(* Logix 5000 project; controller RSL5k_18_Template_noLib Emulate 5570 rev 32.11; software revision 32.02; part 12 of 16 *)
(* tags used below, declared in another part *)
   Inp_SpeedFdbk : REAL;   // Speed Feedbak in Drive Units (typ. 0-32767 = 0 to max freq.)
   Inp_Datalink : REAL;   // Auxiliary Signal (datalink) Input in Drive (raw) Units
   Inp_Ready : BOOL;   // 1=Drive is ready to run
   Inp_Running : BOOL;   // 1=Drive is Running (active)
   Inp_CommandDir : BOOL;   // 1=Drive is commanded Forward, 0=Drive is commanded Reverse
   Inp_ActualDir : BOOL;   // 1=Drive is running Forward, 0=Drive is running Reverse
   Inp_Accelerating : BOOL;   // 1=Drive is accelerating
   Inp_Decelerating : BOOL;   // 1=Drive is decelerating
   Inp_Alarm : BOOL;   // 1=Drive has an Alarm Condition (see drive display or manual)
   Inp_AtSpeed : BOOL;   // 1=Drive is at commanded speed
   Inp_IOFault : BOOL;   // Input Communication Status 0=OK, 1=fail
   Inp_Sim : BOOL;   // 1=Simulate working drive; 0=Start/Stop/ Monitor actual drive
   Inp_OvrdSpeed : REAL;   // Value to set Speed Reference in Override Mode (SpeedRef EU)
   Inp_OvrdOutDatalink : REAL;   // Value to set Output Datalink in Override Mode (OutDatalink EU)
   Inp_HornInh : BOOL;   // 1 = Inhibit audible alert, 0 = Alllow audible alert
   Inp_Reset : BOOL;   // 1=Reset Shed Latches and Cleared Alarms
   Cfg_HasJog : BOOL;   // 1=Drive Jog Command enabled/visible, 0=Drive Jog Command not allowed
   Cfg_AllowLocal : BOOL;   // 1=Allow Local Start/Stop without alarm, 0=Start/Stop from HMI/prog only
   Cfg_HasRunFdbk : BOOL;   // 1=Drive provides feedback signal on Inp_Running when running
   Cfg_UseRunFdbk : BOOL;   // 1=Drive run feedback should be used for failure checking
   Cfg_HasSpeedFdbk : BOOL;   // 1=Drive provides speed feedback on Inp_SpeedFdbk
   Cfg_UseSpeedFdbk : BOOL;   // 1=Drive speed determines running state, 0=state determined by drive Active input bit
   Cfg_HasInpDatalink : BOOL;   // 1=A signal is connected to Inp_Datalink
   Cfg_HasOutDatalink : BOOL;   // 1=A signal is connected to Out_Datalink
   Cfg_HasMoreObj : BOOL;   // 1=Tells HMI an object with more info is available
   Cfg_SetTrack : BOOL;   // 1=Settings track for unselected sources, 0=no tracking
   Cfg_SetTrackOvrdHand : BOOL;   // 1=Prog/Oper/Ext Settings track Override/Hand
   Cfg_OCmdResets : BOOL;   // 1=New drive OCmd resets shed latches and cleared alarms, 0=OCmdReset req'd.
   Cfg_XCmdResets : BOOL;   // 1=New drive XCmd resets shed latches and cleared alarms, 0=XCmdReset req'd.
   Cfg_OvrdPermIntlk : BOOL;   // 1=Override ignores Bypassable Perm/ Intlk; 0=always use Perm/Intlk
   Cfg_SimScaleEU : BOOL;   // 1=In simulation, scale Speed Ref EU to Speed Fdbk EU
   Cfg_SimScaleRaw : BOOL;   // 1=In simulation, scale Speed Ref EU to raw, then raw to Speed Fdbk EU
   Cfg_DecPlcs : DINT;   // Number of decimal places for speed ref/fdbk display (0..6)
   Cfg_InpDLDecPlcs : DINT;   // Number of decimal places for Input Datalink display (0..6)
   Cfg_OutDLDecPlcs : DINT;   // Number of decimal places for Output Datalink display (0..6)
   Cfg_MinSpdRef : REAL;   // Minimum Speed Reference in EU (for limiting)
   Cfg_MaxSpdRef : REAL;   // Maximum Speed Reference in EU (for limiting)
   Cfg_SpeedRefRawMin : REAL;   // Speed Reference Minimum in Drive (raw) Units (for scaling)
   Cfg_SpeedRefRawMax : REAL;   // Speed Reference Maximum in Drive (raw) Units (for scaling)
   Cfg_SpeedRefEUMin : REAL;   // Speed Reference Minimum in Engineering Units (for scaling)
   Cfg_SpeedRefEUMax : REAL;   // Speed Reference Maximum in Engineering Units (for scaling)
   Cfg_SpeedFdbkRawMin : REAL;   // Speed Feedback Minimum in Drive (raw) Units (for scaling)
   Cfg_SpeedFdbkRawMax : REAL;   // Speed Feedback Maximum in Drive (raw) Units (for scaling)
   Cfg_SpeedFdbkEUMin : REAL;   // Speed Feedback Minimum in Engineering Units (for scaling)
   Cfg_SpeedFdbkEUMax : REAL;   // Speed Feedback Maximum in Engineering Units (for scaling)
   Cfg_InpDatalinkRawMin : REAL;   // Input Datalink Minimum in Drive (raw) Units (for scaling)
   Cfg_InpDatalinkRawMax : REAL;   // Input Datalink Maximum in Drive (raw) Units (for scaling)
   Cfg_InpDatalinkEUMin : REAL;   // Input Datalink Minimum in Engineering Units (for scaling)
   Cfg_InpDatalinkEUMax : REAL;   // Input Datalink Maximum in Engineering Units (for scaling)
   Cfg_OutDatalinkMin : REAL;   // Minimum Output Datalink in EU (for limiting)
   Cfg_OutDatalinkMax : REAL;   // Maximum Output Datalink in EU (for limiting)
   Cfg_OutDatalinkRawMin : REAL;   // Output Datalink Minimum in Drive (raw) Units (for scaling)
   Cfg_OutDatalinkRawMax : REAL;   // Output Datalink Maximum in Drive (raw) Units (for scaling)
   Cfg_OutDatalinkEUMin : REAL;   // Output Datalink Minimum in Engineering Units (for scaling)
   Cfg_OutDatalinkEUMax : REAL;   // Output Datalink Maximum in Engineering Units (for scaling)
   Cfg_StartHornT : REAL;   // Time to sound audible on commanded start (sec) (0=disabled)
   Cfg_SimRampT : REAL;   // Time to ramp speed fdbk when in Simulation (sec)
   Cfg_FailToStartT : REAL;   // Time after Start to get Run Feedback before Fault (sec)
   Cfg_FailToStopT : REAL;   // Time after Stop to drop Run Feedback before Fault (sec)
   Cfg_ResetPulseT : REAL;   // Time to pulse Out_Reset to clear drive fault
   Cfg_MaxJogT : REAL;   // Maximum jog time (sec, 0=unlimited)
   Cfg_OperKeep : SINT;   // Oper keeps control in Prog / Ext: .0=Reference, .1=Start/Stop/Fwd/ Rev, .3=OutDatalink
   Cfg_ProgKeep : SINT;   // Prog keeps control in Oper / Ext: .0=Reference, .1=Start/Stop/Fwd/ Rev, .3=OutDatalink
   Cfg_ExtKeep : SINT;   // Ext keeps control in Prog / Oper: .0=Reference, .1=Start/Stop/Fwd/ Rev, .3=OutDatalink
   PSet_SpeedRef : REAL;   // Program Setting of Speed Reference (EU)
   PSet_OutDatalink : REAL;   // Program Setting of Output Datalink (EU)
   PSet_Owner : DINT;   // Program Owner Request ID (non-zero) or Release (zero)
   XSet_SpeedRef : REAL;   // External Setting of Speed Reference (EU)
   XSet_OutDatalink : REAL;   // External Setting of Output Datalink (EU)
   PCmd_Reset : BOOL;   // Program Command to Reset drive fault and all Alarms requiring Reset
   PCmd_FailToStartAck : ALIAS FOR FailToStart.PCmd_Ack;   // Program Command to Acknowledge Fail to Start Alarm
   PCmd_FailToStopAck : ALIAS FOR FailToStop.PCmd_Ack;   // Program Command to Acknowledge Fail to Stop Alarm
   PCmd_IntlkTripAck : ALIAS FOR IntlkTrip.PCmd_Ack;   // Program Command to Acknowledge Interlock Trip Alarm
   PCmd_DriveFaultAck : ALIAS FOR DriveFault.PCmd_Ack;   // Program Command to Acknowledge Drive Fault Alarm
   PCmd_IOFaultAck : ALIAS FOR IOFault.PCmd_Ack;   // Program Command to Acknowledge I/O Fault Alarm
   XCmd_StartFwd : BOOL;   // External Command to Start Drive Forward
   XCmd_StartRev : BOOL;   // External Command to Start Drive Reverse
   XCmd_Stop : BOOL;   // External Command to Stop Drive
   XCmd_JogFwd : BOOL;   // External Command to Jog Drive Forward
   XCmd_JogRev : BOOL;   // External Command to Jog Drive Reverse
   XCmd_Reset : BOOL;   // Ext Cmd to clear shed latches and cleared alarms
   Val_SpeedFdbk : REAL;   // Speed Feedback (actual) from drive
   Val_InpDatalink : REAL;   // Input Datalink value from drive
   Val_SpeedRefEUMin : REAL;   // Minimum of Speed Reference = MIN (Cfg_SpeedFdbkEUMin, Cfg_SpeedFdbkEUMax)
   Val_SpeedRefEUMax : REAL;   // Maximum of Speed Reference = MAX (Cfg_SpeedFdbkEUMin, Cfg_SpeedFdbkEUMax)
   Val_SpeedFdbkEUMin : REAL;   // Minimum of Speed Feedback = MIN (Cfg_SpeedFdbkEUMin, Cfg_SpeedFdbkEUMax)
   Val_SpeedFdbkEUMax : REAL;   // Maximum of Speed Feedback = MAX (Cfg_SpeedFdbkEUMin, Cfg_SpeedFdbkEUMax)
   Val_Fdbk : DINT;   // Device Feedback 0=Stopped, 1=Running Fwd 2=Running Rev 3=Accelerating 4=Decelerating
   Val_Sts : DINT;   // Device Sts: 0=? 1=Stopped 2=RunFwd 3=RunRev 4=RunSlow 5=StartFwd 6=StartRev 7=StartSlow 8=JogFwd 9=JogRev 10=Stopping
   Val_Owner : DINT;   // Current Object Owner ID (0=not owned)
   Sts_CommandDir : BOOL;   // 1=Drive commanded to Forward, 0=Reverse
   Sts_ActualDir : BOOL;   // 1=Drive Actual direction is Forward, 0=Reverse
   Sts_Accel : BOOL;   // 1=Drive is Accelerating
   Sts_Decel : BOOL;   // 1=Drive is Decelerating
   Sts_NotReady : BOOL;   // 1=Drive is Not Ready (cannot be started) Check alarms, stops, faults
   Sts_Alarm : BOOL;   // 1=Drive has an Alarm (see drive display or manual)
   Sts_AtSpeed : BOOL;   // 1=Drive is running at reference speed
   Sts_Bypass : BOOL;   // 1=Bypassable Interlocks and Permissives are Bypassed
   Sts_BypActive : BOOL;   // 1=Bypassing Active (Bypassed or Maintenance)
   Nrdy_CfgErr : BOOL;   // 1=Device Not Ready: Configuration Error
   Nrdy_Fail : BOOL;   // 1=Device Not Ready: Device Failure (Shed Requires Reset)
   Nrdy_IOFault : BOOL;   // 1=Device Not Ready: I/O Fault (Shed Requires Reset)
   Nrdy_PrioStop : BOOL;   // 1=Device Not Ready: Oper/Ext Priority Stop Requires Reset
   Sts_MaintByp : BOOL;   // 1=A Maintenance Bypass is Active, display icon
   Err_Timer : BOOL;   // 1=Error in Config: Invalid Check or Reset Pulse Time (use 0 to 2147483)
   Err_Sim : BOOL;   // 1=Error in Config: simulation timer preset: use 0 to 2147483)
   Err_FdbkRaw : BOOL;   // 1=Erron in Config: Speed Fdbk Raw Min = Max
   Err_FdbkEU : BOOL;   // 1=Error in Config: Speed Fdbk EU Min = Max
   Err_RefLim : BOOL;   // 1=Error in Config: Speed Ref Limit Min > Max
   Err_RefEU : BOOL;   // 1=Error in Config: Speed Ref EU Min = Max
   Err_RefRaw : BOOL;   // 1=Error in Config: Speed Ref Raw Min = Max
   Err_InpDLRaw : BOOL;   // 1=Error in Config: Input Datalink Raw Min = Max
   Err_InpDLEU : BOOL;   // 1=Error in Config: Input Datalink EU Min = Max
   Err_OutDLLim : BOOL;   // 1=Error in Config: Output Datalink Limits Min > Max
   Err_OutDLEU : BOOL;   // 1=Error in Config: Output Datalink EU Min = Max
   Err_OutDLRaw : BOOL;   // 1=Error in Config: Output Datalink Raw Min = Max
   Sts_Hand : ALIAS FOR CmdSrc.Sts_Hand;
   Sts_Maint : ALIAS FOR CmdSrc.Sts_Maint;
   Sts_Ovrd : ALIAS FOR CmdSrc.Sts_Ovrd;
   Sts_Ext : ALIAS FOR CmdSrc.Sts_Ext;
   Sts_Prog : ALIAS FOR CmdSrc.Sts_Prog;
   Sts_Oper : ALIAS FOR CmdSrc.Sts_Oper;
   Sts_RdyAck : BOOL;   // 1=An alarm is ready to be acknowledged
   Sts_FailToStart : ALIAS FOR FailToStart.Inp;   // 1=Drive Failed to Start (One-Shot)
   Sts_FailToStop : ALIAS FOR FailToStop.Inp;   // 1=Drive Failed to Stop
   P_VSD : BOOL;   // Unique Parameter Name for auto - discovery
   CmdSrc : P_CmdSrc;   // Drive Mode Selection
   IOFault : P_Alarm;   // I/O Fault Alarm
   IntlkTrip : P_Alarm;   // Interlock Trip Alarm
   FailToStop : P_Alarm;   // Drive Failed to Stop Alarm
   FailToStart : P_Alarm;   // Drive Failed to Start Alarm
   Cfg_Tag : STRING_20;   // Tagname for display on HMI
   Cfg_Label : STRING_20;   // Label for graphic symbol displayed on HMI
   Cfg_Desc : STRING_40;   // Description for display on HMI
   Wrk_Run : BOOL;   // 1=Drive should be "running", 0=should be "stopped"
   Wrk_StartRetrigT : TIMER;   // Time to pulse start output on start command retrigger (Maint)
   Wrk_StopRetrigT : TIMER;   // Time to pulse stop output on stop command retrigger (Maint)
   Wrk_RunFdbk : BOOL;   // Run Feedback based on mode, simulation, etc. 1=running
   Wrk_Bypass : BOOL;   // Internal Bypassable Permissives and Interlocks are Bypassed flag
   Cfg_SpeedRefEU : STRING_8;   // Speed Reference Engineering Units for display on HMI
   Wrk_SpeedRef : REAL;   // Working copy of Speed Reference (for limiting)
   Wrk_Rev : BOOL;   // Working (internal) Direction 1=Reverse 0=Forward (default)
   Wrk_Jog : BOOL;   // 1=Jog Drive, 0=Drive not jogging
   Wrk_ResetT : TIMER;   // Reset Output Pulse Timer
   Wrk_ResetONS : BOOL;   // One-Shot to fire Reset Timer to ensure min. output ON time.
   Cfg_SpeedFdbkEU : STRING_8;   // Speed Feedback Engineering Units for display on HMI
   Cfg_OutDatalinkLabel : STRING_20;   // Datalink Output Label displayed on faceplate
   Cfg_InpDatalinkLabel : STRING_20;   // Datalink Input Label displayed on faceplate
   Cfg_OutDatalinkEU : STRING_8;   // Datalink Output Engineering Units for display on HMI
   Cfg_InpDatalinkEU : STRING_8;   // Datalink Input Engineering Units for display on HMI
   Wrk_OutDatalink : REAL;   // Selected Output Datalink setting
   Cfg_RevText : STRING_16;   // Name for Reverse Direction, e.g., "Down", "Reverse"
   Cfg_FwdText : STRING_16;   // Name for Forward Direction, e.g., "Up", "Forward"
   Wrk_StopT : TIMER;   // Stop Check Timer (for Fail to Stop)
   Wrk_StartT : TIMER;   // Start Check Timer (for Fail to Start)
   Wrk_Step : REAL;   // Amount to change simulated Speed Fdbk this scan (ramp)
   Wrk_ScanTime : REAL;   // Seconds since previous scan
   Wrk_ScanT : TIMER;   // Scan Timer (milliseconds, always runs)
   Wrk_SimFdbkTgt : REAL;   // Speed Ref converted to Speed Fdbk units for simulation: target speed fdbk
   HMI_Type : STRING_16;   // Type identifier for HMI navigation
   Wrk_JogT : TIMER;   // Jog Timer
   Wrk_OperKeep3ONS : BOOL;   // Oper Keep bit 3 one-shot store
   Wrk_OperKeep1ONS : BOOL;   // Oper Keep bit 1 one-shot store
   Wrk_OperKeep0ONS : BOOL;   // Oper Keep bit 0 one-shot store
   Wrk_ProgKeep3ONS : BOOL;   // Prog Keep bit 3 one-shot store
   Wrk_ProgKeep1ONS : BOOL;   // Prog Keep bit 1 one-shot store
   Wrk_ProgKeep0ONS : BOOL;   // Prog Keep bit 0 one-shot store
   HMI_Lib : STRING_12;   // Display Library for Faceplate call-up
   Wrk_SimScaleEUONS : BOOL;   // Cfg_SimScaleEU became true this scan
   Wrk_SimScaleRawONS : BOOL;   // Cfg_SimScaleRaw became true this scan
   Wrk_StartInhT : TIMER;   // Local Start Inhibit Timer
   Wrk_StopInhT : TIMER;   // Local Stop Inhibit Timer
   Wrk_NoLongerSim : BOOL;   // Switched from Simulated to Real Drive this scan
   Wrk_Hand : BOOL;   // Perform Hand Mode alignment with actual device state
   Cfg_Area : STRING_Area;   // Process Area for security
   Wrk_StartHornT : TIMER;   // Timer for audible alert or start
   OCmd_ResetAckAll : BOOL;   // Oper Cmd to reset shed latches and cleared alarms, plus Acknowledge alarms
   OCmd_Reset : BOOL;   // Oper Cmd to clear shed latches and cleared alarms
   OCmd_JogRev : BOOL;   // Operator Command to Jog Drive Reverse (not cleared by instruction!)
   OCmd_JogFwd : BOOL;   // Operator Command to Jog Drive Forward (not cleared by instruction!)
   OCmd_Stop : BOOL;   // Operator Command to Stop Drive
   OCmd_StartRev : BOOL;   // Operator Command to Start Drive Reverse
   OCmd_StartFwd : BOOL;   // Operator Command to Start Drive Forward
   MCmd_Check : BOOL;   // Maintenance Command to Check (not bypass) all Interlocks and Permissives
   MCmd_Bypass : BOOL;   // Maintenance Command to Bypass all Bypassable Interlocks and Permissives
   OSet_OutDatalink : REAL;   // Operator Setting of Output Datalink (EU)
   OSet_SpeedRef : REAL;   // Operator Setting of Speed Reference (EU)
   ORdy_OSet : BOOL;   // 1=Ready for OSets (other than Speed Ref) (enables data entry fields)
   ORdy_SpeedRef : BOOL;   // 1=Ready for OSet_SpeedRef (enables data entry field)
   MRdy_Check : BOOL;   // 1=Ready for MCmd_Check (enables HMI button)
   MRdy_Bypass : BOOL;   // 1=Ready for MCmd_Bypass (enables HMI button)
   Wrk_ExtKeep3ONS : BOOL;   // Ext Keep bit 3 one-shot store
   Wrk_ExtKeep1ONS : BOOL;   // Ext Keep bit 1 one-shot store
   Wrk_ExtKeep0ONS : BOOL;   // Ext Keep bit 0 one-shot store
   Wrk_ExtHas3 : BOOL;   // External has Output Datalink
   Wrk_ExtHas1 : BOOL;   // External has Commands
   Wrk_ExtHas0 : BOOL;   // External has Speed Reference
   Wrk_ProgHas3 : BOOL;   // Program has Output Datalink
   Wrk_ProgHas1 : BOOL;   // Program has Commands
   Wrk_ProgHas0 : BOOL;   // Program has Speed Reference
   Wrk_OperHas3 : BOOL;   // Operator has Output Datalink
   Wrk_OperHas1 : BOOL;   // Operator has Commands
   Wrk_OperHas0 : BOOL;   // Operator has Speed Reference
(* P_VSD, continued *)

ROUTINE Logic   (* ladder *)
// Normal Scan: control / monitor Variable-Speed Drive
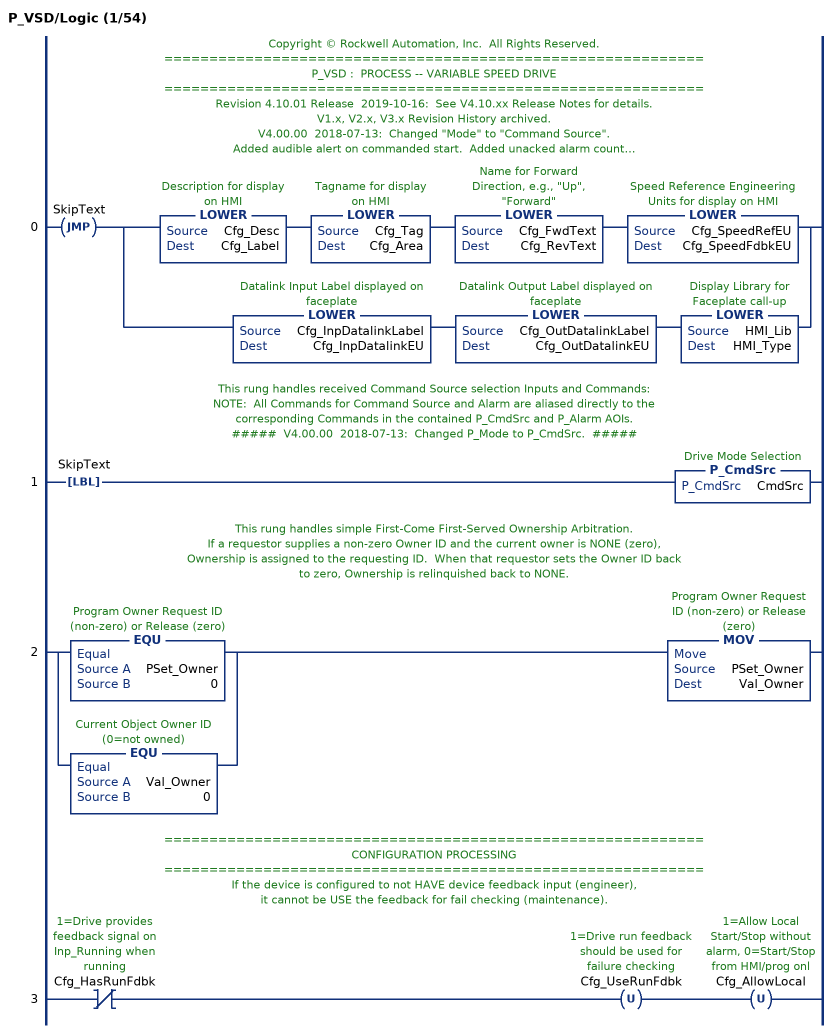
   // Copyright © Rockwell Automation, Inc.  All Rights Reserved.
   // ============================================================
   // P_VSD :  PROCESS -- VARIABLE SPEED DRIVE
   // ============================================================
   // Revision 4.10.01 Release  2019-10-16:  See V4.10.xx Release Notes for details.
   // V1.x, V2.x, V3.x Revision History archived.
   // V4.00.00  2018-07-13:  Changed "Mode" to "Command Source".
   // Added audible alert on commanded start.  Added unacked alarm count.
   // Changed Inf_ items to HMI_, and added Cfg_Area for security.
   // Changed Start / Stop / Fwd / Rev / Jog to StartFwd / StartRev /Stop / JogFwd / JogRev.
   // Deleted Cfg_PCmdClear; all Program Commands are now self-clearing.
   // All OCmds/MCmds and ORdys/MRdys are now Local Tags.
   // Added Sts_RdyAck and Sts_ResetReqd for use by external objects.
   // Aligned ready bit naming with command bit names.
   // Added configurable decimal places for display on HMI.
   // Modifications to Output Datalink clamp limit restrictions / checking.
   // Changed delay / time configuration items to REAL seconds.
   // Updated Val_Sts to common enumeration across all motors and drives.
   // V4.00.02  2018-10-30:  Corrected handling Allow Local when horn is enabled
   // V4.10.00  2019-03-25:  Changed availability to use input availability from interlocks.
   // Added Horn Status, Horn Inhibit. Updated to P_CmdSrc V4.10.00.
   // Modified simulated run feedback to handle run at zero speed ref.
   // Added Cfg_HasMoreObj.
   // V4.10.01  2019-10-16:  Corrected handling of Start Horn on shed conditions.
   // Modified to lock out jog when jog time expires until jog commands
   // are cleared. Modified to handle overlapping Horn and Jog times.
   // ============================================================
   // This Instruction controls and monitors a Variable-Speed Drive (AC or DC) and provides:
   // *  Starting, stopping, jogging of drive, setting speed reference and direction
   // *  Monitoring of run feedback, display of actual drive status, including accel, decel, direction, speed
   // *  Detection of Failure to Start, Failure to Stop, Drive Fault
   // *  Monitoring of Permissive conditions to allow starting
   // * Monitoring of Interlock conditions to stop / prevent starting
   // * Simulation, providing feedback of a working drive while disabling outputs
   // * Monitoring of I/O communication faults
   // * Alarms for Fail to Start, Fail to Stop, Interlock Trip, Drive Fault, I/O Fault
   // * Option to automatically reset faults and alarms when operator commands
   // motor to start or stop
   // * Supports HMI "breadcrumbs" for Alarm Inhibited, Bad Configuration,
   // Not Ready, Maintenance Bypass Active
   // * "Available" status for use by automation logic to know whether motor
   // can be controlled by other objects.
   // * Horn output for audible alert prior to starting motor.
   // Command Sources are arbitrated by a P_CmdSrc Add-On Instruction instance.
   // Command Sources: Operator, External, Program, External, Override, Maintenance,
   // Out of Service, Hand.  Alarms are provided by P_Alarm Add-On Instruction instances.
   // ============================================================
   // SHOW LOCAL STRINGS
   // ============================================================
   // The STRINGs containing the text associated with each instance of this
   // instruction cannot be Input or Output Parameters, because STRINGs are not
   //  'atomic' types. (Inputs and Outputs must be SINT, INT, DINT, REAL, or BOOL.)
   // In order to make it easier to find and configure these STRINGs, this rung
   // was added.  THE JMP (and the LBL on the following rung)
   // MUST NOT BE REMOVED!!!
   // To view the STRINGs, go to the instruction instance (in LD or FBD), RIGHT-click
   // to bring up the context menu and select "Open Instruction Logic".
   // This rung will appear with the STRING values for the selected instance.
   // You may double-click the STRING values here to modify them as well.
   // #####  V4.00.00  2018-07-13:  Added string for Cfg_Area, renamed Inf_* to HMI_*.  #####
   0: JMP(SkipText)[LOWER(Cfg_Desc,Cfg_Label) LOWER(Cfg_Tag,Cfg_Area) LOWER(Cfg_FwdText,Cfg_RevText) LOWER(Cfg_SpeedRefEU,Cfg_SpeedFdbkEU) ,LOWER(Cfg_InpDatalinkLabel,Cfg_InpDatalinkEU) LOWER(Cfg_OutDatalinkLabel,Cfg_OutDatalinkEU) LOWER(HMI_Lib,HMI_Type) ];
   // This rung handles received Command Source selection Inputs and Commands:
   // NOTE:  All Commands for Command Source and Alarm are aliased directly to the
   // corresponding Commands in the contained P_CmdSrc and P_Alarm AOIs.
   // #####  V4.00.00  2018-07-13:  Changed P_Mode to P_CmdSrc.  #####
   1: LBL(SkipText)P_CmdSrc(CmdSrc);
   // This rung handles simple First-Come First-Served Ownership Arbitration.
   // If a requestor supplies a non-zero Owner ID and the current owner is NONE (zero),
   // Ownership is assigned to the requesting ID.  When that requestor sets the Owner ID back
   // to zero, Ownership is relinquished back to NONE.
   2: [EQU(PSet_Owner,0) ,EQU(Val_Owner,0) ]MOV(PSet_Owner,Val_Owner);
   // ============================================================
   // CONFIGURATION PROCESSING
   // ============================================================
   // If the device is configured to not HAVE device feedback input (engineer),
   // it cannot be USE the feedback for fail checking (maintenance).
   3: XIO(Cfg_HasRunFdbk)OTU(Cfg_UseRunFdbk)OTU(Cfg_AllowLocal);
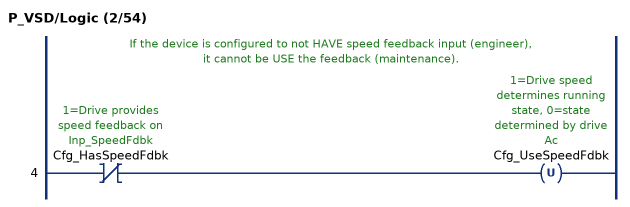
   // If the device is configured to not HAVE speed feedback input (engineer),
   // it cannot be USE the feedback (maintenance).
   4: XIO(Cfg_HasSpeedFdbk)OTU(Cfg_UseSpeedFdbk);
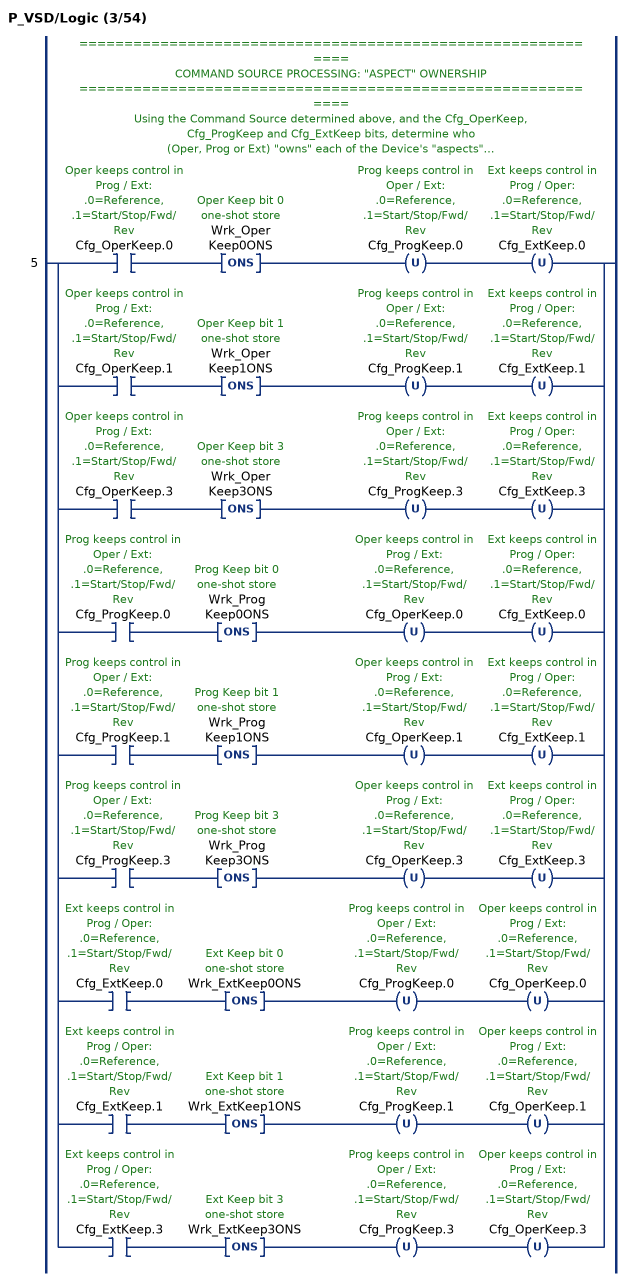
   // ============================================================
   // COMMAND SOURCE PROCESSING: "ASPECT" OWNERSHIP
   // ============================================================
   // Using the Command Source determined above, and the Cfg_OperKeep,
   // Cfg_ProgKeep and Cfg_ExtKeep bits, determine who
   // (Oper, Prog or Ext) "owns" each of the Device's "aspects":
   // Speed Reference (.0), Start/Stop (.1), and Output Datalink (.3).
   // The bits within Cfg_OperKeep, Cfg_ProgKeep and Cfg_ExtKeep determine
   // which "aspects" (sub-functions of this AOI) are retained by the Operator,
   // by the Program, or by the External command source when either of the
   // other command sources is selected.
   // All aspects (functions) may be "kept" (basically locking the Oper/Prog/Ext
   // selections, rendering the Command Source selection moot.
   // (You get to explain how it works to your operators!!!).
   // However, it is NOT allowed to have any given aspect "kept" by more than
   // one source.  This rung ensures that no aspect is "kept" by multiple sources.
   // #####  V4.00.00  2018-07-13:  Using P_CmdSrc, added External command source.  #####
   5: [XIC(Cfg_OperKeep.0) ONS(Wrk_OperKeep0ONS) OTU(Cfg_ProgKeep.0) OTU(Cfg_ExtKeep.0) ,XIC(Cfg_OperKeep.1) ONS(Wrk_OperKeep1ONS) OTU(Cfg_ProgKeep.1) OTU(Cfg_ExtKeep.1) ,XIC(Cfg_OperKeep.3) ONS(Wrk_OperKeep3ONS) OTU(Cfg_ProgKeep.3) OTU(Cfg_ExtKeep.3) ,XIC(Cfg_ProgKeep.0) ONS(Wrk_ProgKeep0ONS) OTU(Cfg_OperKeep.0) OTU(Cfg_ExtKeep.0) ,XIC(Cfg_ProgKeep.1) ONS(Wrk_ProgKeep1ONS) OTU(Cfg_OperKeep.1) OTU(Cfg_ExtKeep.1) ,XIC(Cfg_ProgKeep.3) ONS(Wrk_ProgKeep3ONS) OTU(Cfg_OperKeep.3) OTU(Cfg_ExtKeep.3) ,XIC(Cfg_ExtKeep.0) ONS(Wrk_ExtKeep0ONS) OTU(Cfg_ProgKeep.0) OTU(Cfg_OperKeep.0) ,XIC(Cfg_ExtKeep.1) ONS(Wrk_ExtKeep1ONS) OTU(Cfg_ProgKeep.1) OTU(Cfg_OperKeep.1) ,XIC(Cfg_ExtKeep.3) ONS(Wrk_ExtKeep3ONS) OTU(Cfg_ProgKeep.3) OTU(Cfg_OperKeep.3) ];
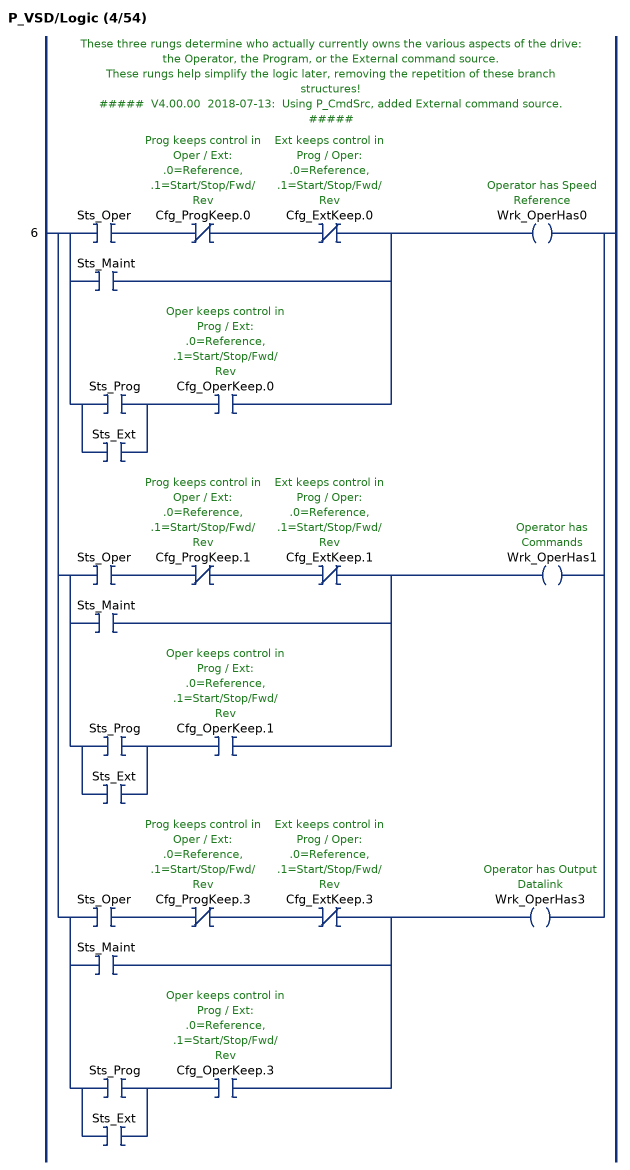
   // These three rungs determine who actually currently owns the various aspects of the drive:
   // the Operator, the Program, or the External command source.
   // These rungs help simplify the logic later, removing the repetition of these branch structures!
   // #####  V4.00.00  2018-07-13:  Using P_CmdSrc, added External command source.  #####
   6: [[XIC(Sts_Oper) XIO(Cfg_ProgKeep.0) XIO(Cfg_ExtKeep.0) ,XIC(Sts_Maint) ,[XIC(Sts_Prog) ,XIC(Sts_Ext) ] XIC(Cfg_OperKeep.0) ] OTE(Wrk_OperHas0) ,[XIC(Sts_Oper) XIO(Cfg_ProgKeep.1) XIO(Cfg_ExtKeep.1) ,XIC(Sts_Maint) ,[XIC(Sts_Prog) ,XIC(Sts_Ext) ] XIC(Cfg_OperKeep.1) ] OTE(Wrk_OperHas1) ,[XIC(Sts_Oper) XIO(Cfg_ProgKeep.3) XIO(Cfg_ExtKeep.3) ,XIC(Sts_Maint) ,[XIC(Sts_Prog) ,XIC(Sts_Ext) ] XIC(Cfg_OperKeep.3) ] OTE(Wrk_OperHas3) ];
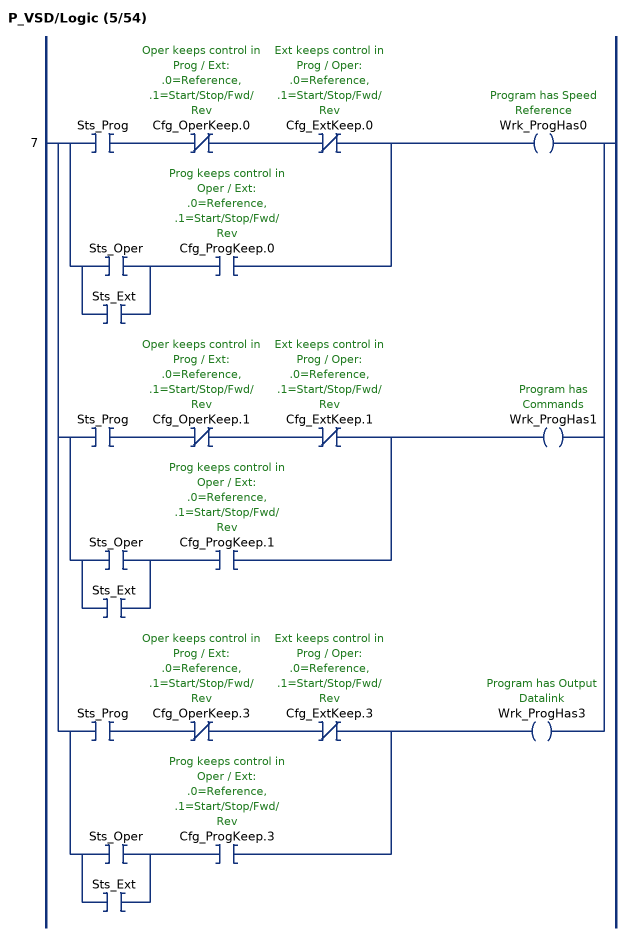
   7: [[XIC(Sts_Prog) XIO(Cfg_OperKeep.0) XIO(Cfg_ExtKeep.0) ,[XIC(Sts_Oper) ,XIC(Sts_Ext) ] XIC(Cfg_ProgKeep.0) ] OTE(Wrk_ProgHas0) ,[XIC(Sts_Prog) XIO(Cfg_OperKeep.1) XIO(Cfg_ExtKeep.1) ,[XIC(Sts_Oper) ,XIC(Sts_Ext) ] XIC(Cfg_ProgKeep.1) ] OTE(Wrk_ProgHas1) ,[XIC(Sts_Prog) XIO(Cfg_OperKeep.3) XIO(Cfg_ExtKeep.3) ,[XIC(Sts_Oper) ,XIC(Sts_Ext) ] XIC(Cfg_ProgKeep.3) ] OTE(Wrk_ProgHas3) ];
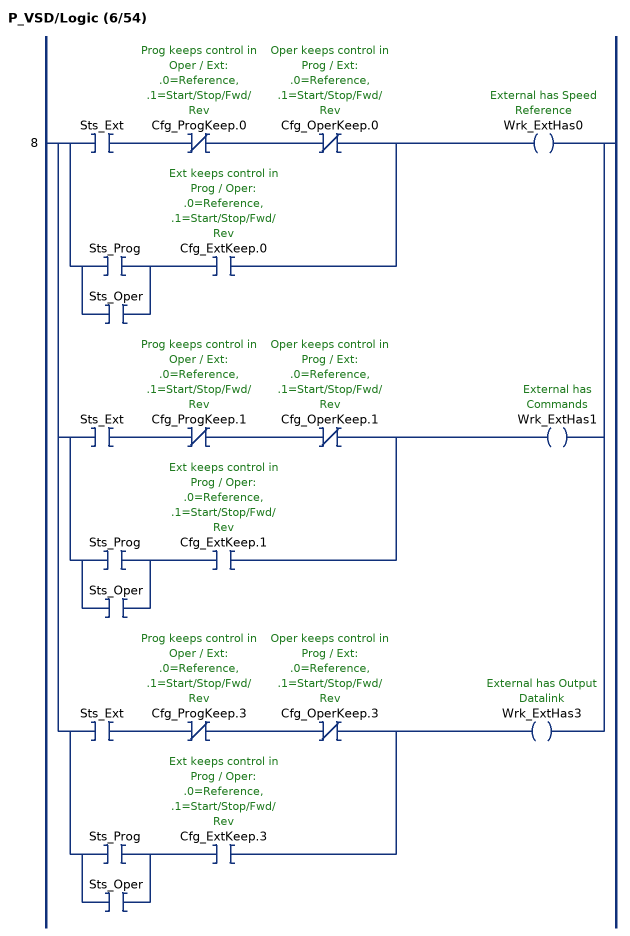
   8: [[XIC(Sts_Ext) XIO(Cfg_ProgKeep.0) XIO(Cfg_OperKeep.0) ,[XIC(Sts_Prog) ,XIC(Sts_Oper) ] XIC(Cfg_ExtKeep.0) ] OTE(Wrk_ExtHas0) ,[XIC(Sts_Ext) XIO(Cfg_ProgKeep.1) XIO(Cfg_OperKeep.1) ,[XIC(Sts_Prog) ,XIC(Sts_Oper) ] XIC(Cfg_ExtKeep.1) ] OTE(Wrk_ExtHas1) ,[XIC(Sts_Ext) XIO(Cfg_ProgKeep.3) XIO(Cfg_OperKeep.3) ,[XIC(Sts_Prog) ,XIC(Sts_Oper) ] XIC(Cfg_ExtKeep.3) ] OTE(Wrk_ExtHas3) ];
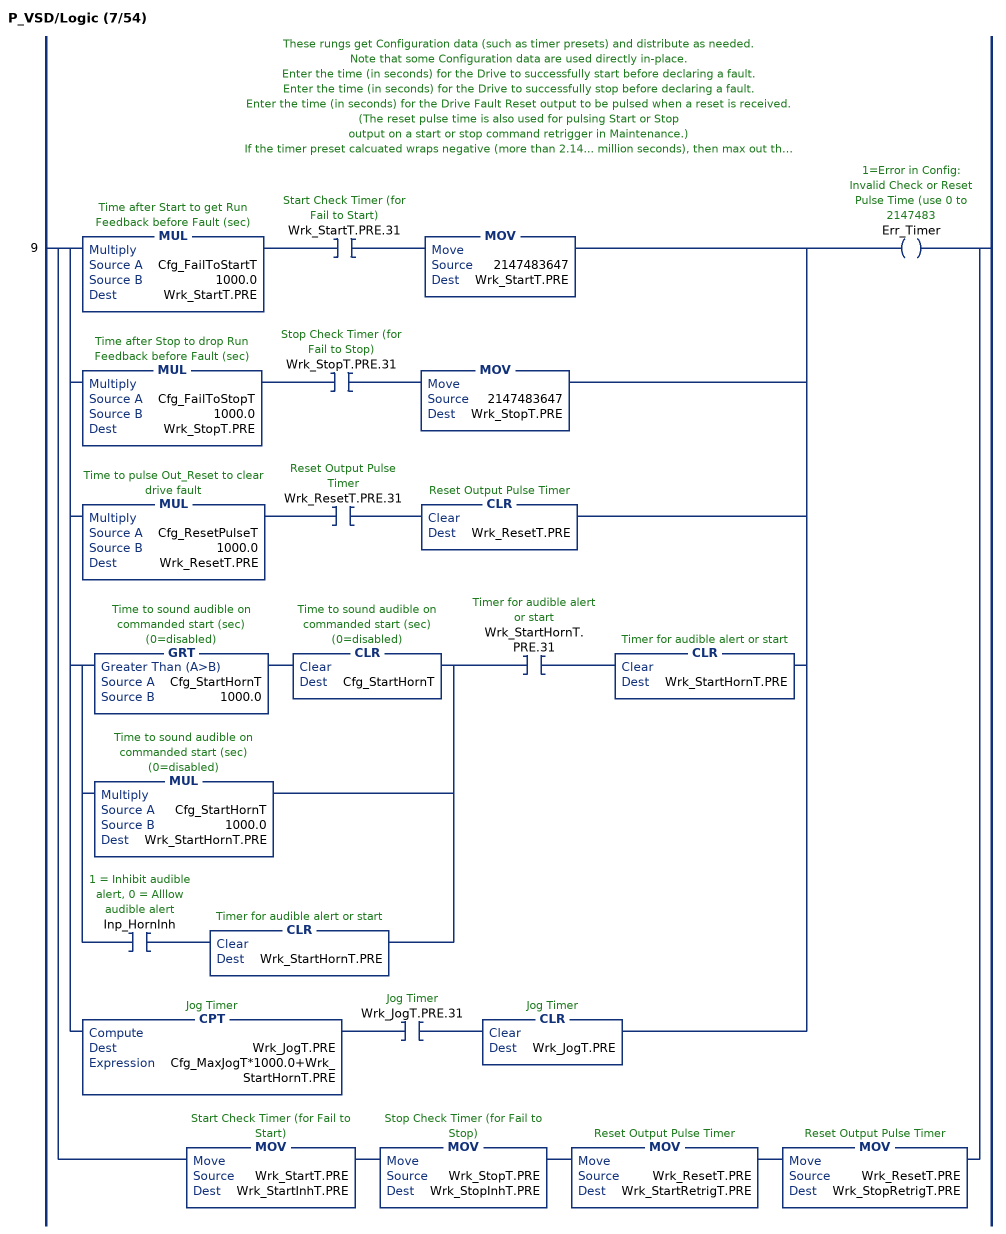
   // These rungs get Configuration data (such as timer presets) and distribute as needed.
   // Note that some Configuration data are used directly in-place.
   // Enter the time (in seconds) for the Drive to successfully start before declaring a fault.
   // Enter the time (in seconds) for the Drive to successfully stop before declaring a fault.
   // Enter the time (in seconds) for the Drive Fault Reset output to be pulsed when a reset is received.
   // (The reset pulse time is also used for pulsing Start or Stop
   // output on a start or stop command retrigger in Maintenance.)
   // If the timer preset calcuated wraps negative (more than 2.14... million seconds), then max out the
   // or clear the Timer Preset (as appropriate) and flag it.  Note that a negative timer preset will fault the controller!!!
   // #####  V4.00.00  2018-07-13:  Added audible alert prior to commanded start.  #####
   // #####  Changed delay / time configuration items to REAL seconds.  #####
   // #####  V4.10.00  2019-03-25:  Added Inp_HornInh to disable Horn operation.  #####
   // #####  V4.10.01  2019-10-16:  Modified to handle overlapping Horn and Jog times.  #####
   9: [[MUL(Cfg_FailToStartT,1000.0,Wrk_StartT.PRE) XIC(Wrk_StartT.PRE.31) MOV(2147483647,Wrk_StartT.PRE) ,MUL(Cfg_FailToStopT,1000.0,Wrk_StopT.PRE) XIC(Wrk_StopT.PRE.31) MOV(2147483647,Wrk_StopT.PRE) ,MUL(Cfg_ResetPulseT,1000.0,Wrk_ResetT.PRE) XIC(Wrk_ResetT.PRE.31) CLR(Wrk_ResetT.PRE) ,[GRT(Cfg_StartHornT,1000.0) CLR(Cfg_StartHornT) ,MUL(Cfg_StartHornT,1000.0,Wrk_StartHornT.PRE) ,XIC(Inp_HornInh) CLR(Wrk_StartHornT.PRE) ] XIC(Wrk_StartHornT.PRE.31) CLR(Wrk_StartHornT.PRE) ,CPT(Wrk_JogT.PRE,Cfg_MaxJogT*1000.0+Wrk_StartHornT.PRE) XIC(Wrk_JogT.PRE.31) CLR(Wrk_JogT.PRE) ] OTE(Err_Timer) ,MOV(Wrk_StartT.PRE,Wrk_StartInhT.PRE) MOV(Wrk_StopT.PRE,Wrk_StopInhT.PRE) MOV(Wrk_ResetT.PRE,Wrk_StartRetrigT.PRE) MOV(Wrk_ResetT.PRE,Wrk_StopRetrigT.PRE) ];
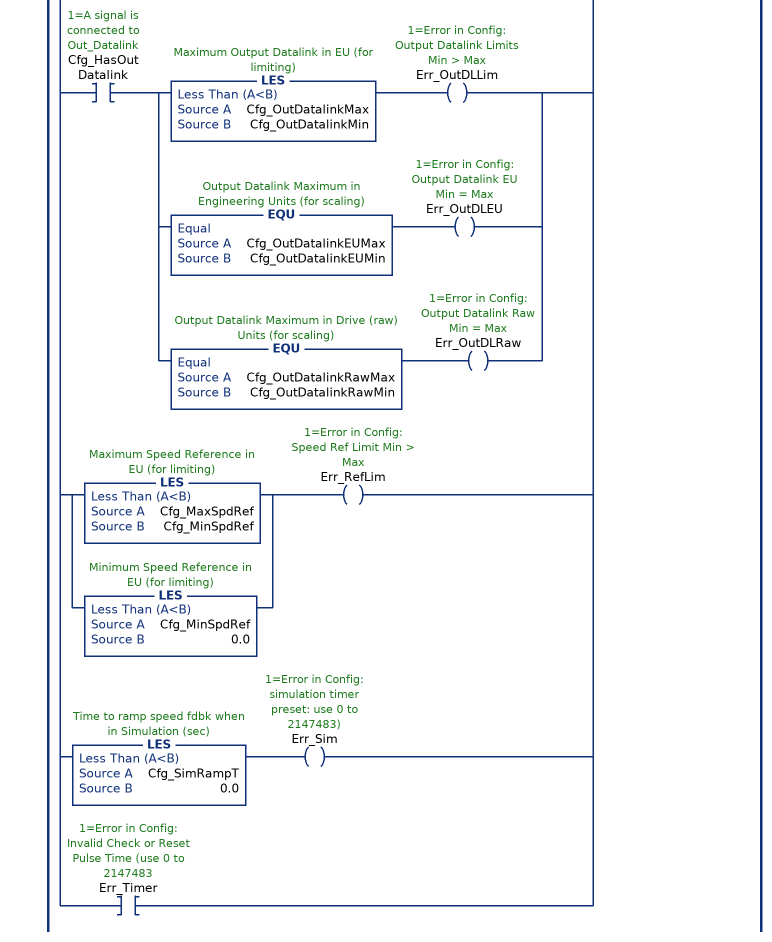
   // This rung handles the reports of all Bad Configuration Status.
   // Individual bits are provided for various status:
   // Bad Raw Scaling configs
   // Bad Engineering Units Scaling configs
   // Bad Min or Max Speed Reference clamp limit
   // Bad simulation speed ramp time
   // Bad timer config from (rung above)
   // Bad Alarm config (from P_Alarm)
   // Bad Cfg_OperKeep / Cfg_ProgKeep config
   // Then a summary Bad Config status is provided, simply an OR of the individual bits.
   // #####  V4.00.00  2018-07-13:  Modified to allow the special case where min and max clamping  #####
   // #####  limits (speed or output datalink) can be EQUAL (clamp at a specific value).  #####
   // #####  Changed delay / time configuration items to REAL seconds.  #####
   10: [XIC(Cfg_HasSpeedFdbk) [EQU(Cfg_SpeedFdbkRawMax,Cfg_SpeedFdbkRawMin) OTE(Err_FdbkRaw) ,EQU(Cfg_SpeedFdbkEUMax,Cfg_SpeedFdbkEUMin) OTE(Err_FdbkEU) ] ,EQU(Cfg_SpeedRefEUMax,Cfg_SpeedRefEUMin) OTE(Err_RefEU) ,EQU(Cfg_SpeedRefRawMax,Cfg_SpeedRefRawMin) OTE(Err_RefRaw) ,XIC(Cfg_HasInpDatalink) [EQU(Cfg_InpDatalinkRawMax,Cfg_InpDatalinkRawMin) OTE(Err_InpDLRaw) ,EQU(Cfg_InpDatalinkEUMax,Cfg_InpDatalinkEUMin) OTE(Err_InpDLEU) ] ,XIC(Cfg_HasOutDatalink) [LES(Cfg_OutDatalinkMax,Cfg_OutDatalinkMin) OTE(Err_OutDLLim) ,EQU(Cfg_OutDatalinkEUMax,Cfg_OutDatalinkEUMin) OTE(Err_OutDLEU) ,EQU(Cfg_OutDatalinkRawMax,Cfg_OutDatalinkRawMin) OTE(Err_OutDLRaw) ] ,[LES(Cfg_MaxSpdRef,Cfg_MinSpdRef) ,LES(Cfg_MinSpdRef,0.0) ] OTE(Err_RefLim) ,LES(Cfg_SimRampT,0.0) OTE(Err_Sim) ,XIC(Err_Timer) ]OTE(Nrdy_CfgErr);
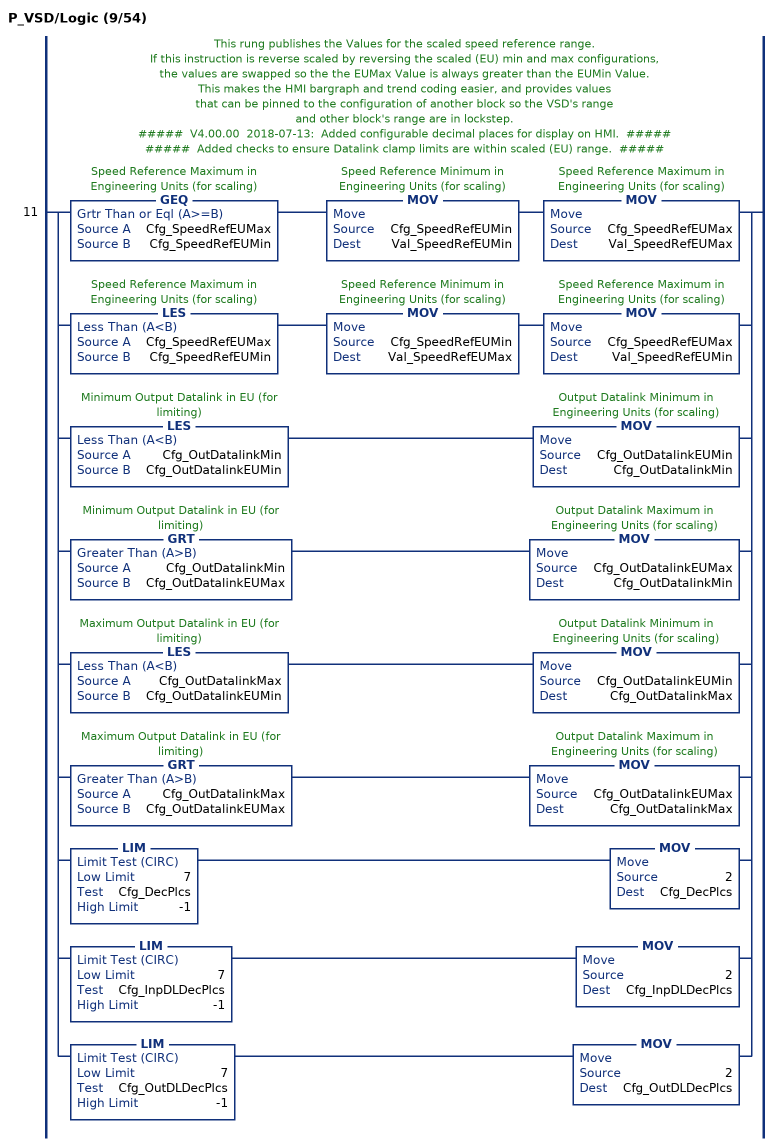
   // This rung publishes the Values for the scaled speed reference range.
   // If this instruction is reverse scaled by reversing the scaled (EU) min and max configurations,
   // the values are swapped so the the EUMax Value is always greater than the EUMin Value.
   // This makes the HMI bargraph and trend coding easier, and provides values
   // that can be pinned to the configuration of another block so the VSD's range
   //  and other block's range are in lockstep.
   // #####  V4.00.00  2018-07-13:  Added configurable decimal places for display on HMI.  #####
   // #####  Added checks to ensure Datalink clamp limits are within scaled (EU) range.  #####
   11: [GEQ(Cfg_SpeedRefEUMax,Cfg_SpeedRefEUMin) MOV(Cfg_SpeedRefEUMin,Val_SpeedRefEUMin) MOV(Cfg_SpeedRefEUMax,Val_SpeedRefEUMax) ,LES(Cfg_SpeedRefEUMax,Cfg_SpeedRefEUMin) MOV(Cfg_SpeedRefEUMin,Val_SpeedRefEUMax) MOV(Cfg_SpeedRefEUMax,Val_SpeedRefEUMin) ,LES(Cfg_OutDatalinkMin,Cfg_OutDatalinkEUMin) MOV(Cfg_OutDatalinkEUMin,Cfg_OutDatalinkMin) ,GRT(Cfg_OutDatalinkMin,Cfg_OutDatalinkEUMax) MOV(Cfg_OutDatalinkEUMax,Cfg_OutDatalinkMin) ,LES(Cfg_OutDatalinkMax,Cfg_OutDatalinkEUMin) MOV(Cfg_OutDatalinkEUMin,Cfg_OutDatalinkMax) ,GRT(Cfg_OutDatalinkMax,Cfg_OutDatalinkEUMax) MOV(Cfg_OutDatalinkEUMax,Cfg_OutDatalinkMax) ,LIM(7,Cfg_DecPlcs,-1) MOV(2,Cfg_DecPlcs) ,LIM(7,Cfg_InpDLDecPlcs,-1) MOV(2,Cfg_InpDLDecPlcs) ,LIM(7,Cfg_OutDLDecPlcs,-1) MOV(2,Cfg_OutDLDecPlcs) ];
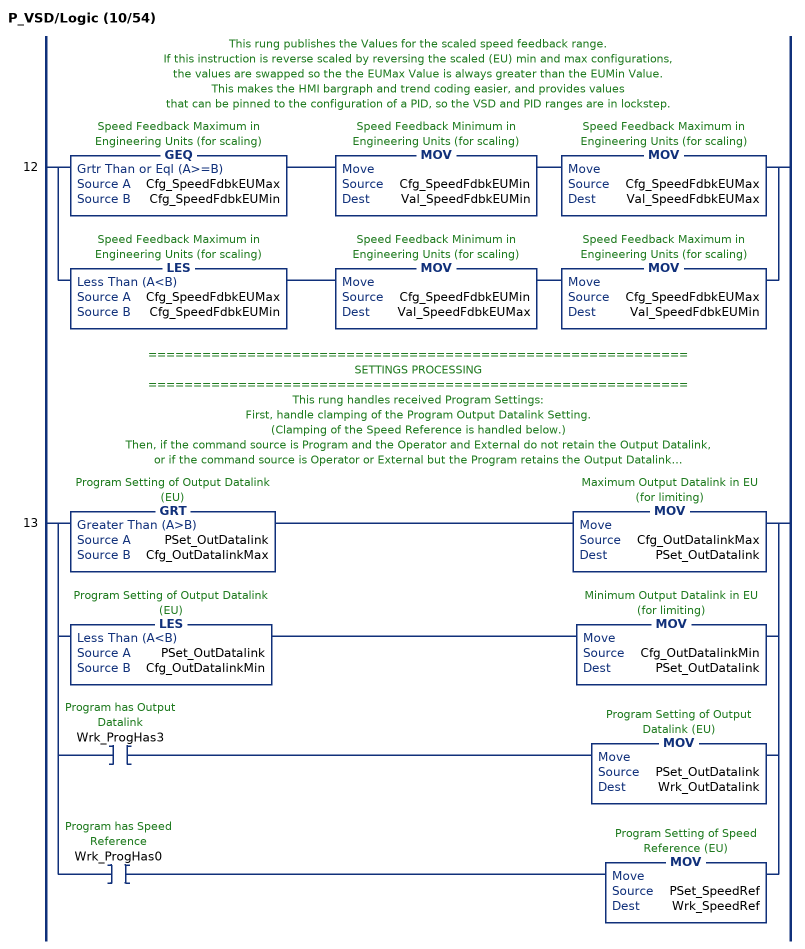
   // This rung publishes the Values for the scaled speed feedback range.
   // If this instruction is reverse scaled by reversing the scaled (EU) min and max configurations,
   // the values are swapped so the the EUMax Value is always greater than the EUMin Value.
   // This makes the HMI bargraph and trend coding easier, and provides values
   // that can be pinned to the configuration of a PID, so the VSD and PID ranges are in lockstep.
   12: [GEQ(Cfg_SpeedFdbkEUMax,Cfg_SpeedFdbkEUMin) MOV(Cfg_SpeedFdbkEUMin,Val_SpeedFdbkEUMin) MOV(Cfg_SpeedFdbkEUMax,Val_SpeedFdbkEUMax) ,LES(Cfg_SpeedFdbkEUMax,Cfg_SpeedFdbkEUMin) MOV(Cfg_SpeedFdbkEUMin,Val_SpeedFdbkEUMax) MOV(Cfg_SpeedFdbkEUMax,Val_SpeedFdbkEUMin) ];
   // ============================================================
   // SETTINGS PROCESSING
   // ============================================================
   // This rung handles received Program Settings:
   // First, handle clamping of the Program Output Datalink Setting.
   // (Clamping of the Speed Reference is handled below.)
   // Then, if the command source is Program and the Operator and External do not retain the Output Datalink,
   // or if the command source is Operator or External but the Program retains the Output Datalink,
   // use the Program Setting for the Output Datalink.
   // The Program Setting for the Speed Reference is handled similarly.
   // #####  Changed P_Mode to P_CmdSrc. Added External Command Source and Commands.  #####
   13: [GRT(PSet_OutDatalink,Cfg_OutDatalinkMax) MOV(Cfg_OutDatalinkMax,PSet_OutDatalink) ,LES(PSet_OutDatalink,Cfg_OutDatalinkMin) MOV(Cfg_OutDatalinkMin,PSet_OutDatalink) ,XIC(Wrk_ProgHas3) MOV(PSet_OutDatalink,Wrk_OutDatalink) ,XIC(Wrk_ProgHas0) MOV(PSet_SpeedRef,Wrk_SpeedRef) ];
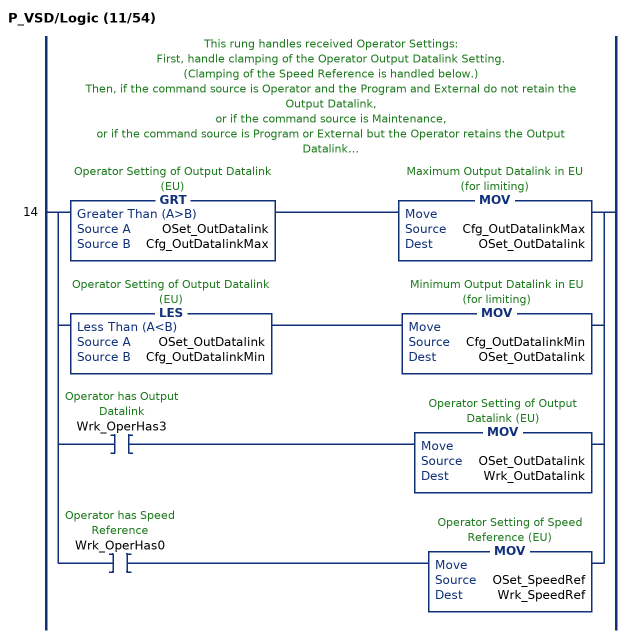
   // This rung handles received Operator Settings:
   // First, handle clamping of the Operator Output Datalink Setting.
   // (Clamping of the Speed Reference is handled below.)
   // Then, if the command source is Operator and the Program and External do not retain the Output Datalink,
   // or if the command source is Maintenance,
   // or if the command source is Program or External but the Operator retains the Output Datalink,
   // use the Operator Setting for the Output Datalink.
   // The Operator Setting for the Speed Reference is handled similarly.
   // #####  Changed P_Mode to P_CmdSrc. Added External Command Source and Commands.  #####
   14: [GRT(OSet_OutDatalink,Cfg_OutDatalinkMax) MOV(Cfg_OutDatalinkMax,OSet_OutDatalink) ,LES(OSet_OutDatalink,Cfg_OutDatalinkMin) MOV(Cfg_OutDatalinkMin,OSet_OutDatalink) ,XIC(Wrk_OperHas3) MOV(OSet_OutDatalink,Wrk_OutDatalink) ,XIC(Wrk_OperHas0) MOV(OSet_SpeedRef,Wrk_SpeedRef) ];
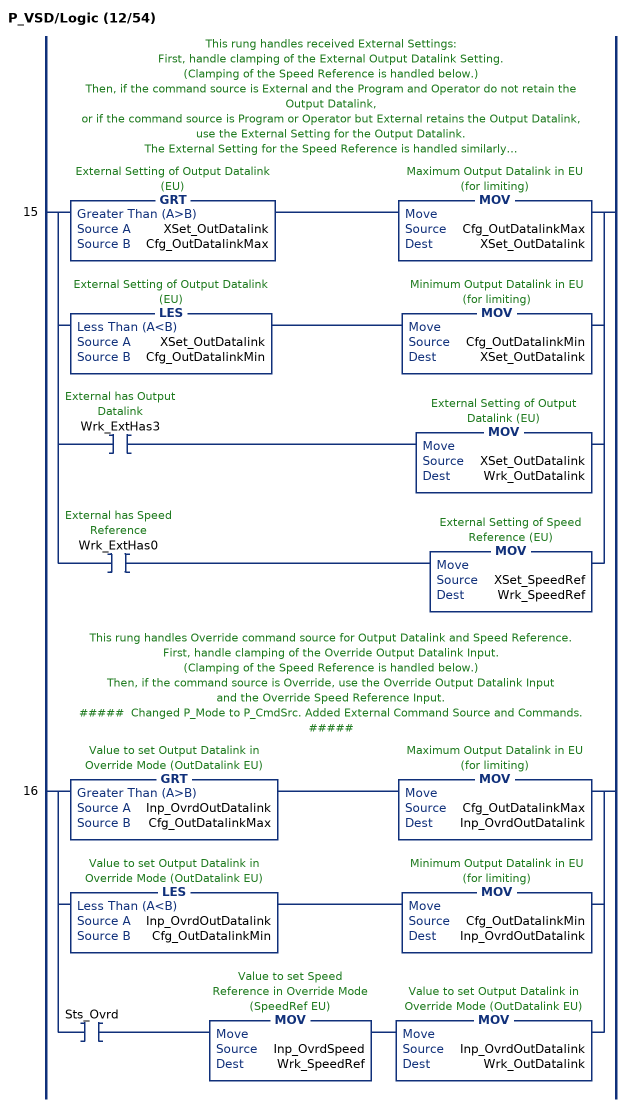
   // This rung handles received External Settings:
   // First, handle clamping of the External Output Datalink Setting.
   // (Clamping of the Speed Reference is handled below.)
   // Then, if the command source is External and the Program and Operator do not retain the Output Datalink,
   // or if the command source is Program or Operator but External retains the Output Datalink,
   // use the External Setting for the Output Datalink.
   // The External Setting for the Speed Reference is handled similarly.
   // #####  Changed P_Mode to P_CmdSrc. Added External Command Source and Commands.  #####
   15: [GRT(XSet_OutDatalink,Cfg_OutDatalinkMax) MOV(Cfg_OutDatalinkMax,XSet_OutDatalink) ,LES(XSet_OutDatalink,Cfg_OutDatalinkMin) MOV(Cfg_OutDatalinkMin,XSet_OutDatalink) ,XIC(Wrk_ExtHas3) MOV(XSet_OutDatalink,Wrk_OutDatalink) ,XIC(Wrk_ExtHas0) MOV(XSet_SpeedRef,Wrk_SpeedRef) ];
   // This rung handles Override command source for Output Datalink and Speed Reference.
   // First, handle clamping of the Override Output Datalink Input.
   // (Clamping of the Speed Reference is handled below.)
   // Then, if the command source is Override, use the Override Output Datalink Input
   // and the Override Speed Reference Input.
   // #####  Changed P_Mode to P_CmdSrc. Added External Command Source and Commands.  #####
   16: [GRT(Inp_OvrdOutDatalink,Cfg_OutDatalinkMax) MOV(Cfg_OutDatalinkMax,Inp_OvrdOutDatalink) ,LES(Inp_OvrdOutDatalink,Cfg_OutDatalinkMin) MOV(Cfg_OutDatalinkMin,Inp_OvrdOutDatalink) ,XIC(Sts_Ovrd) MOV(Inp_OvrdSpeed,Wrk_SpeedRef) MOV(Inp_OvrdOutDatalink,Wrk_OutDatalink) ];
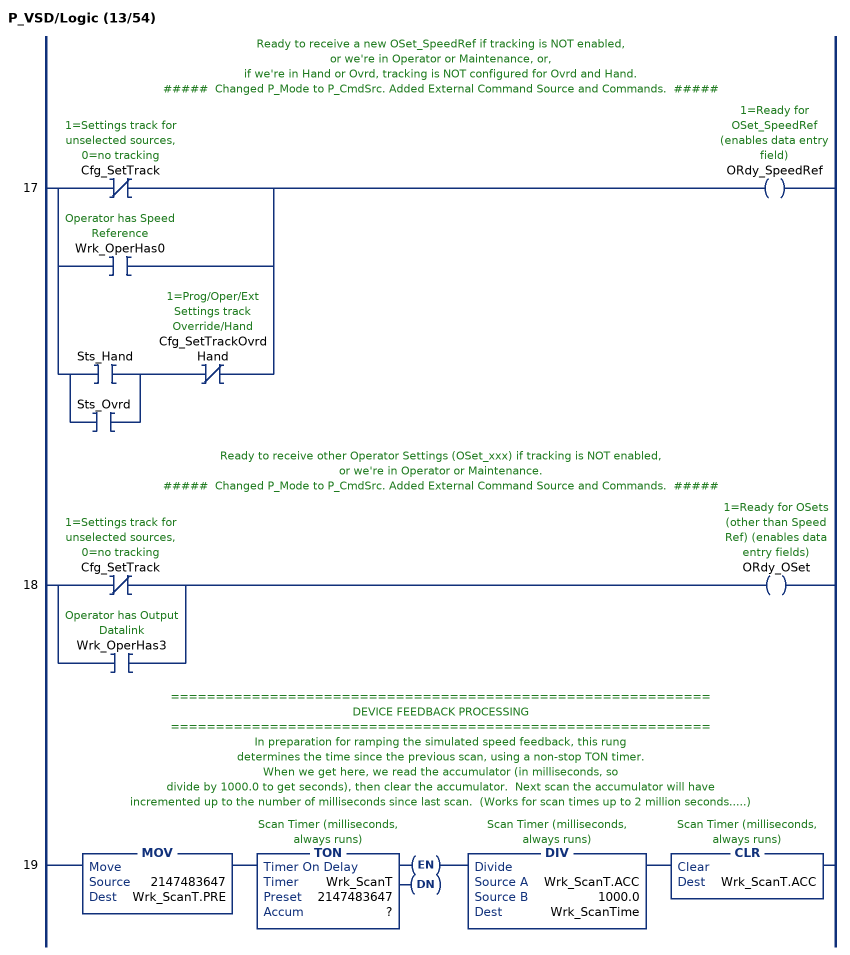
   // Ready to receive a new OSet_SpeedRef if tracking is NOT enabled,
   // or we're in Operator or Maintenance, or,
   // if we're in Hand or Ovrd, tracking is NOT configured for Ovrd and Hand.
   // #####  Changed P_Mode to P_CmdSrc. Added External Command Source and Commands.  #####
   17: [XIO(Cfg_SetTrack) ,XIC(Wrk_OperHas0) ,[XIC(Sts_Hand) ,XIC(Sts_Ovrd) ] XIO(Cfg_SetTrackOvrdHand) ]OTE(ORdy_SpeedRef);
   // Ready to receive other Operator Settings (OSet_xxx) if tracking is NOT enabled,
   // or we're in Operator or Maintenance.
   // #####  Changed P_Mode to P_CmdSrc. Added External Command Source and Commands.  #####
   18: [XIO(Cfg_SetTrack) ,XIC(Wrk_OperHas3) ]OTE(ORdy_OSet);
   // ============================================================
   // DEVICE FEEDBACK PROCESSING
   // ============================================================
   // In preparation for ramping the simulated speed feedback, this rung
   // determines the time since the previous scan, using a non-stop TON timer.
   // When we get here, we read the accumulator (in milliseconds, so
   // divide by 1000.0 to get seconds), then clear the accumulator.  Next scan the accumulator will have
   // incremented up to the number of milliseconds since last scan.  (Works for scan times up to 2 million seconds.....)
   19: MOV(2147483647,Wrk_ScanT.PRE)TON(Wrk_ScanT,?,?)DIV(Wrk_ScanT.ACC,1000.0,Wrk_ScanTime)CLR(Wrk_ScanT.ACC);
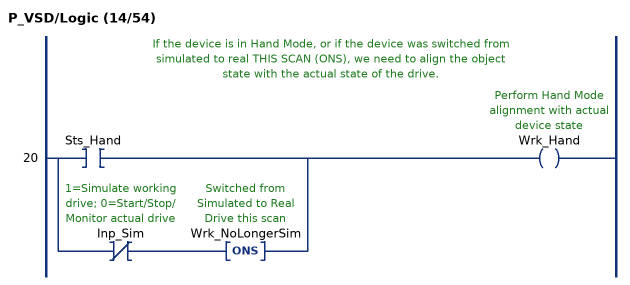
   // If the device is in Hand Mode, or if the device was switched from
   // simulated to real THIS SCAN (ONS), we need to align the object
   // state with the actual state of the drive.
   20: [XIC(Sts_Hand) ,XIO(Inp_Sim) ONS(Wrk_NoLongerSim) ]OTE(Wrk_Hand);
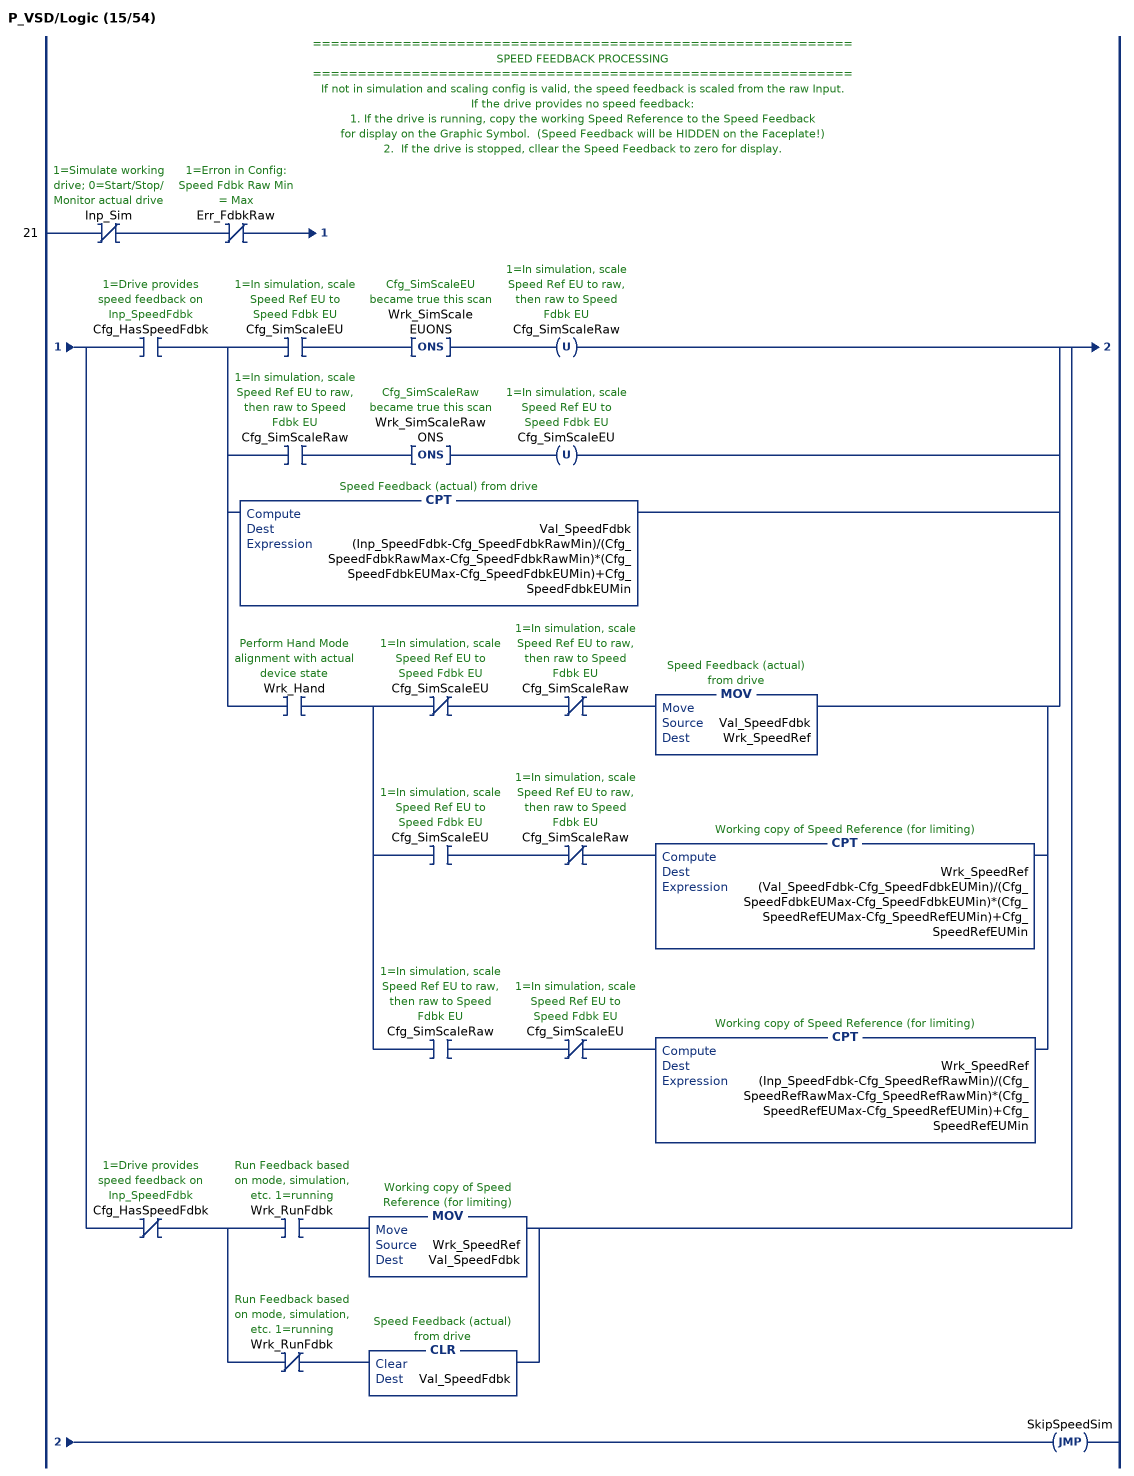
   // ============================================================
   // SPEED FEEDBACK PROCESSING
   // ============================================================
   // If not in simulation and scaling config is valid, the speed feedback is scaled from the raw Input.
   // If the drive provides no speed feedback:
   // 1. If the drive is running, copy the working Speed Reference to the Speed Feedback
   // for display on the Graphic Symbol.  (Speed Feedback will be HIDDEN on the Faceplate!)
   // 2.  If the drive is stopped, cllear the Speed Feedback to zero for display.
   21: XIO(Inp_Sim)XIO(Err_FdbkRaw)[XIC(Cfg_HasSpeedFdbk) [XIC(Cfg_SimScaleEU) ONS(Wrk_SimScaleEUONS) OTU(Cfg_SimScaleRaw) ,XIC(Cfg_SimScaleRaw) ONS(Wrk_SimScaleRawONS) OTU(Cfg_SimScaleEU) ,CPT(Val_SpeedFdbk,(Inp_SpeedFdbk-Cfg_SpeedFdbkRawMin)/(Cfg_SpeedFdbkRawMax-Cfg_SpeedFdbkRawMin)*(Cfg_SpeedFdbkEUMax-Cfg_SpeedFdbkEUMin)+Cfg_SpeedFdbkEUMin) ,XIC(Wrk_Hand) [XIO(Cfg_SimScaleEU) XIO(Cfg_SimScaleRaw) MOV(Val_SpeedFdbk,Wrk_SpeedRef) ,XIC(Cfg_SimScaleEU) XIO(Cfg_SimScaleRaw) CPT(Wrk_SpeedRef,(Val_SpeedFdbk-Cfg_SpeedFdbkEUMin)/(Cfg_SpeedFdbkEUMax-Cfg_SpeedFdbkEUMin)*(Cfg_SpeedRefEUMax-Cfg_SpeedRefEUMin)+Cfg_SpeedRefEUMin) ,XIC(Cfg_SimScaleRaw) XIO(Cfg_SimScaleEU) CPT(Wrk_SpeedRef,(Inp_SpeedFdbk-Cfg_SpeedRefRawMin)/(Cfg_SpeedRefRawMax-Cfg_SpeedRefRawMin)*(Cfg_SpeedRefEUMax-Cfg_SpeedRefEUMin)+Cfg_SpeedRefEUMin) ] ] ,XIO(Cfg_HasSpeedFdbk) [XIC(Wrk_RunFdbk) MOV(Wrk_SpeedRef,Val_SpeedFdbk) ,XIO(Wrk_RunFdbk) CLR(Val_SpeedFdbk) ] ]JMP(SkipSpeedSim);
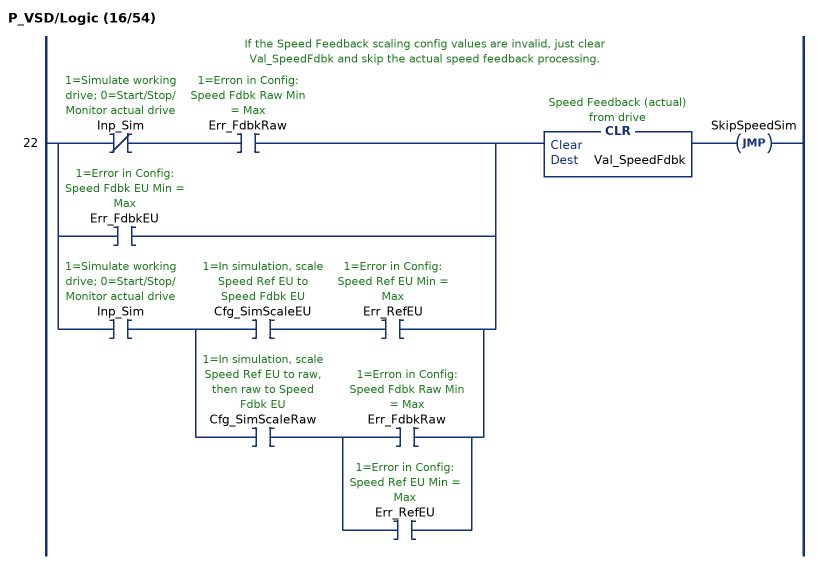
   // If the Speed Feedback scaling config values are invalid, just clear
   // Val_SpeedFdbk and skip the actual speed feedback processing.
   22: [XIO(Inp_Sim) XIC(Err_FdbkRaw) ,XIC(Err_FdbkEU) ,XIC(Inp_Sim) [XIC(Cfg_SimScaleEU) XIC(Err_RefEU) ,XIC(Cfg_SimScaleRaw) [XIC(Err_FdbkRaw) ,XIC(Err_RefEU) ] ] ]CLR(Val_SpeedFdbk)JMP(SkipSpeedSim);
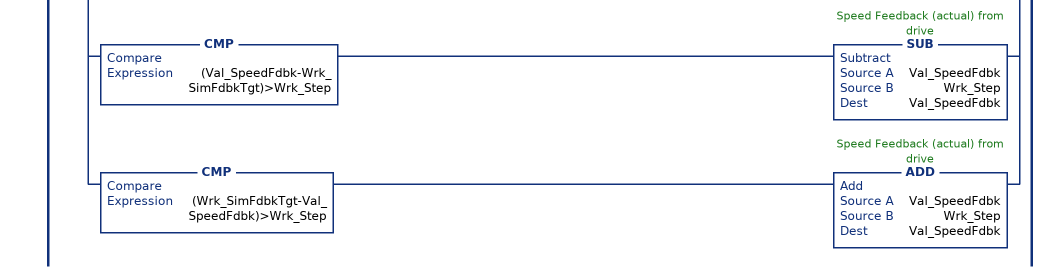
   // If in simulation, simulate accel/decel.
   // #####  V4.00.00  2018-07-13:  Changed delay / time configuration items to REAL seconds.  #####
   23: XIC(Inp_Sim)[[XIC(Wrk_Run) ,XIC(Wrk_Jog) ] [XIO(Cfg_SimScaleEU) XIO(Cfg_SimScaleRaw) MOV(Wrk_SpeedRef,Wrk_SimFdbkTgt) ,[XIC(Cfg_SimScaleEU) XIO(Cfg_SimScaleRaw) CPT(Wrk_SimFdbkTgt,(Wrk_SpeedRef-Cfg_SpeedRefEUMin)/(Cfg_SpeedRefEUMax-Cfg_SpeedRefEUMin)*(Cfg_SpeedFdbkEUMax-Cfg_SpeedFdbkEUMin)+Cfg_SpeedFdbkEUMin) ,XIC(Cfg_SimScaleRaw) [CPT(Wrk_SimFdbkTgt,(Wrk_SpeedRef-Cfg_SpeedRefEUMin)/(Cfg_SpeedRefEUMax-Cfg_SpeedRefEUMin)*(Cfg_SpeedRefRawMax-Cfg_SpeedRefRawMin)+Cfg_SpeedRefRawMin) ,CPT(Wrk_SimFdbkTgt,(Wrk_SimFdbkTgt-Cfg_SpeedFdbkRawMin)/(Cfg_SpeedFdbkRawMax-Cfg_SpeedFdbkRawMin)*(Cfg_SpeedFdbkEUMax-Cfg_SpeedFdbkEUMin)+Cfg_SpeedFdbkEUMin) ] ] ] ,[XIO(Wrk_Run) XIO(Wrk_Jog) ,XIO(Wrk_Rev) XIO(Sts_ActualDir) ,XIC(Wrk_Rev) XIC(Sts_ActualDir) ] CLR(Wrk_SimFdbkTgt) ,GRT(Cfg_SimRampT,0.0) [CPT(Wrk_Step,Cfg_MaxSpdRef/Cfg_SimRampT*Wrk_ScanTime) ,XIC(Cfg_SimScaleEU) XIO(Cfg_SimScaleRaw) CPT(Wrk_Step,(Wrk_Step-Cfg_SpeedRefEUMin)/(Cfg_SpeedRefEUMax-Cfg_SpeedRefEUMin)*(Cfg_SpeedFdbkEUMax-Cfg_SpeedFdbkEUMin)+Cfg_SpeedFdbkEUMin) ,XIC(Cfg_SimScaleRaw) [CPT(Wrk_Step,(Wrk_Step-Cfg_SpeedRefEUMin)/(Cfg_SpeedRefEUMax-Cfg_SpeedRefEUMin)*(Cfg_SpeedRefRawMax-Cfg_SpeedRefRawMin)+Cfg_SpeedRefRawMin) ,CPT(Wrk_Step,(Wrk_Step-Cfg_SpeedFdbkRawMin)/(Cfg_SpeedFdbkRawMax-Cfg_SpeedFdbkRawMin)*(Cfg_SpeedFdbkEUMax-Cfg_SpeedFdbkEUMin)+Cfg_SpeedFdbkEUMin) ] ] ,LEQ(Cfg_SimRampT,0.0) MOV(1.50000000e+038,Wrk_Step) ,CMP(ABS(Val_SpeedFdbk-Wrk_SimFdbkTgt)<=Wrk_Step) MOV(Wrk_SimFdbkTgt,Val_SpeedFdbk) ,CMP((Val_SpeedFdbk-Wrk_SimFdbkTgt)>Wrk_Step) SUB(Val_SpeedFdbk,Wrk_Step,Val_SpeedFdbk) ,CMP((Wrk_SimFdbkTgt-Val_SpeedFdbk)>Wrk_Step) ADD(Val_SpeedFdbk,Wrk_Step,Val_SpeedFdbk) ];
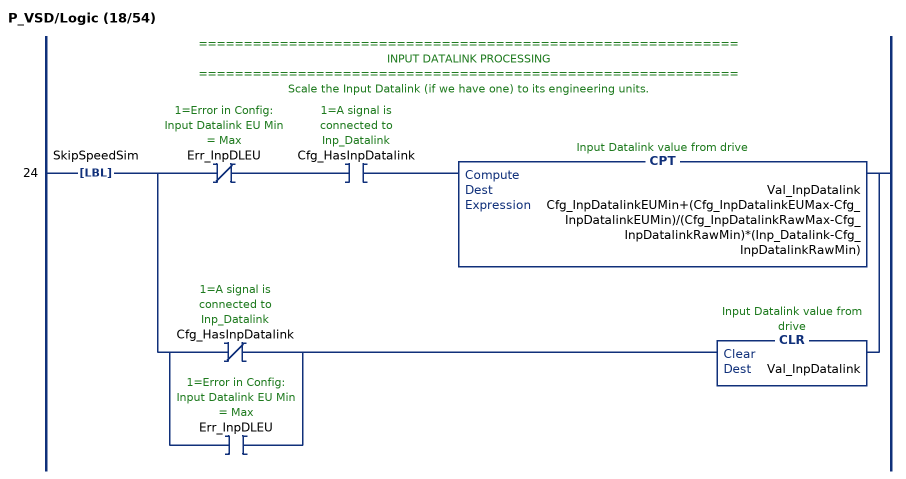
   // ============================================================
   // INPUT DATALINK PROCESSING
   // ============================================================
   // Scale the Input Datalink (if we have one) to its engineering units.
   24: LBL(SkipSpeedSim)[XIO(Err_InpDLEU) XIC(Cfg_HasInpDatalink) CPT(Val_InpDatalink,Cfg_InpDatalinkEUMin+(Cfg_InpDatalinkEUMax-Cfg_InpDatalinkEUMin)/(Cfg_InpDatalinkRawMax-Cfg_InpDatalinkRawMin)*(Inp_Datalink-Cfg_InpDatalinkRawMin)) ,[XIO(Cfg_HasInpDatalink) ,XIC(Err_InpDLEU) ] CLR(Val_InpDatalink) ];
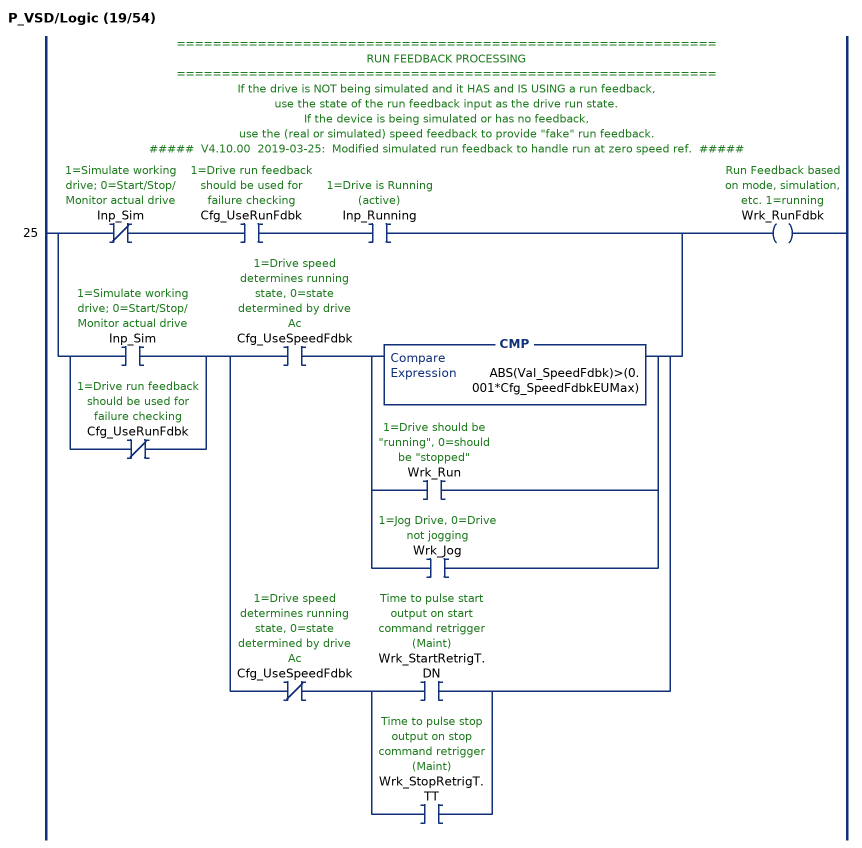
   // ============================================================
   // RUN FEEDBACK PROCESSING
   // ============================================================
   // If the drive is NOT being simulated and it HAS and IS USING a run feedback,
   // use the state of the run feedback input as the drive run state.
   // If the device is being simulated or has no feedback,
   // use the (real or simulated) speed feedback to provide "fake" run feedback.
   // #####  V4.10.00  2019-03-25:  Modified simulated run feedback to handle run at zero speed ref.  #####
   25: [XIO(Inp_Sim) XIC(Cfg_UseRunFdbk) XIC(Inp_Running) ,[XIC(Inp_Sim) ,XIO(Cfg_UseRunFdbk) ] [XIC(Cfg_UseSpeedFdbk) [CMP(ABS(Val_SpeedFdbk)>(0.001*Cfg_SpeedFdbkEUMax)) ,XIC(Wrk_Run) ,XIC(Wrk_Jog) ] ,XIO(Cfg_UseSpeedFdbk) [XIC(Wrk_StartRetrigT.DN) ,XIC(Wrk_StopRetrigT.TT) ] ] ]OTE(Wrk_RunFdbk);
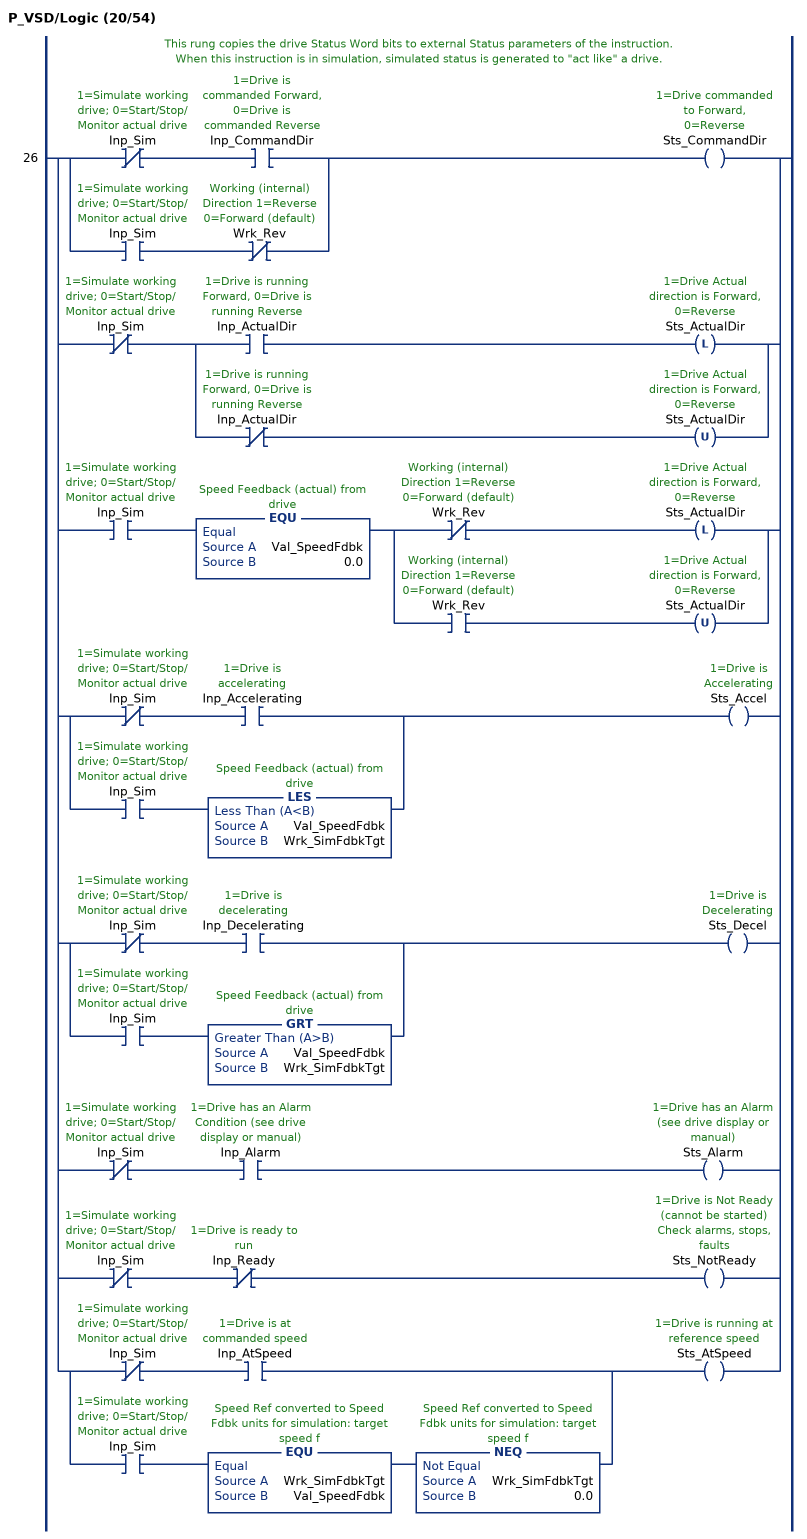
   // This rung copies the drive Status Word bits to external Status parameters of the instruction.
   // When this instruction is in simulation, simulated status is generated to "act like" a drive.
   26: [[XIO(Inp_Sim) XIC(Inp_CommandDir) ,XIC(Inp_Sim) XIO(Wrk_Rev) ] OTE(Sts_CommandDir) ,[XIO(Inp_Sim) [XIC(Inp_ActualDir) OTL(Sts_ActualDir) ,XIO(Inp_ActualDir) OTU(Sts_ActualDir) ] ,XIC(Inp_Sim) EQU(Val_SpeedFdbk,0.0) [XIO(Wrk_Rev) OTL(Sts_ActualDir) ,XIC(Wrk_Rev) OTU(Sts_ActualDir) ] ] ,[XIO(Inp_Sim) XIC(Inp_Accelerating) ,XIC(Inp_Sim) LES(Val_SpeedFdbk,Wrk_SimFdbkTgt) ] OTE(Sts_Accel) ,[XIO(Inp_Sim) XIC(Inp_Decelerating) ,XIC(Inp_Sim) GRT(Val_SpeedFdbk,Wrk_SimFdbkTgt) ] OTE(Sts_Decel) ,XIO(Inp_Sim) XIC(Inp_Alarm) OTE(Sts_Alarm) ,XIO(Inp_Sim) XIO(Inp_Ready) OTE(Sts_NotReady) ,[XIO(Inp_Sim) XIC(Inp_AtSpeed) ,XIC(Inp_Sim) EQU(Wrk_SimFdbkTgt,Val_SpeedFdbk) NEQ(Wrk_SimFdbkTgt,0.0) ] OTE(Sts_AtSpeed) ];
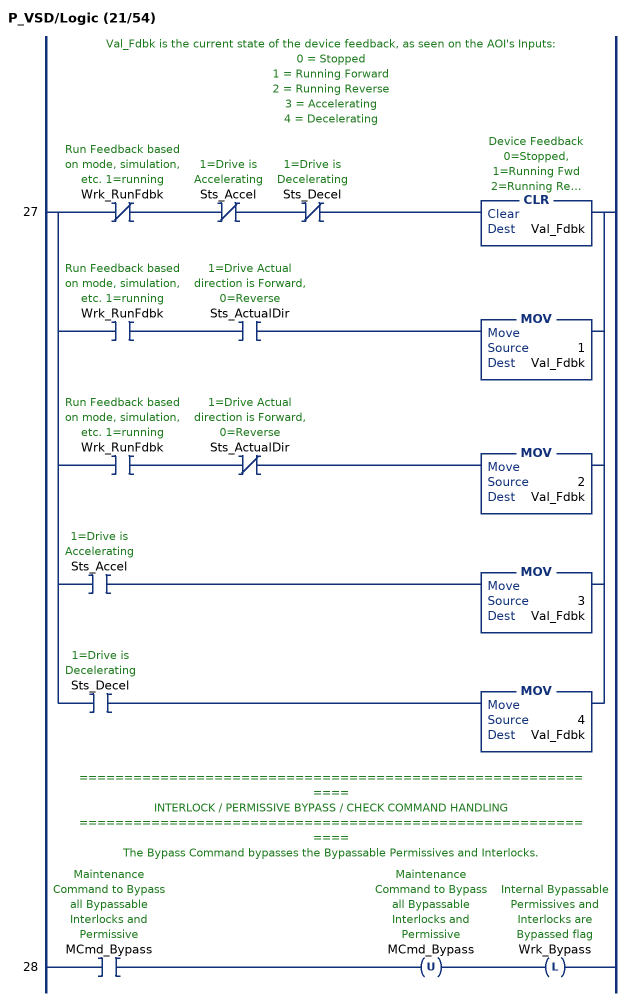
   // Val_Fdbk is the current state of the device feedback, as seen on the AOI's Inputs:
   // 0 = Stopped
   // 1 = Running Forward
   // 2 = Running Reverse
   // 3 = Accelerating
   // 4 = Decelerating
   27: [XIO(Wrk_RunFdbk) XIO(Sts_Accel) XIO(Sts_Decel) CLR(Val_Fdbk) ,XIC(Wrk_RunFdbk) XIC(Sts_ActualDir) MOV(1,Val_Fdbk) ,XIC(Wrk_RunFdbk) XIO(Sts_ActualDir) MOV(2,Val_Fdbk) ,XIC(Sts_Accel) MOV(3,Val_Fdbk) ,XIC(Sts_Decel) MOV(4,Val_Fdbk) ];
   // ============================================================
   // INTERLOCK / PERMISSIVE BYPASS / CHECK COMMAND HANDLING
   // ============================================================
   // The Bypass Command bypasses the Bypassable Permissives and Interlocks.
   28: XIC(MCmd_Bypass)OTU(MCmd_Bypass)OTL(Wrk_Bypass);
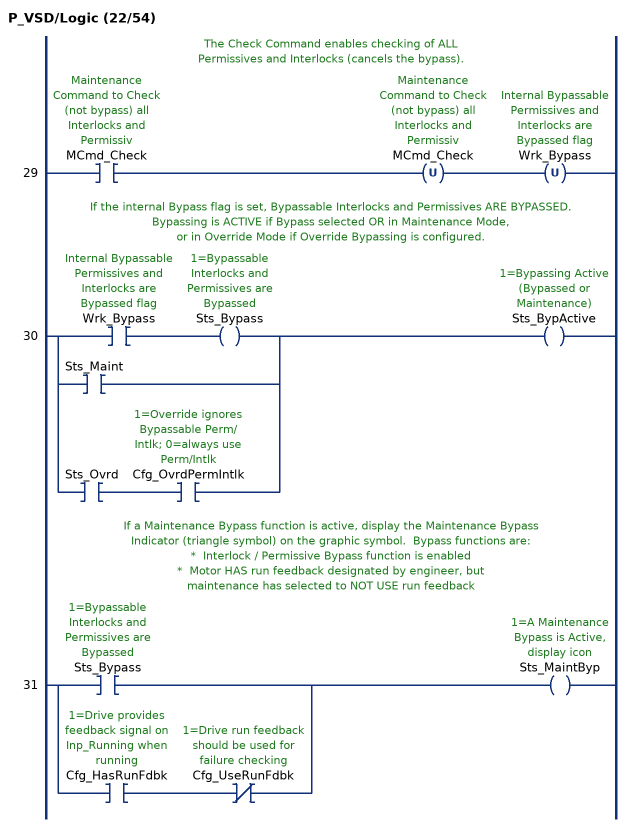
   // The Check Command enables checking of ALL
   // Permissives and Interlocks (cancels the bypass).
   29: XIC(MCmd_Check)OTU(MCmd_Check)OTU(Wrk_Bypass);
   // If the internal Bypass flag is set, Bypassable Interlocks and Permissives ARE BYPASSED.
   // Bypassing is ACTIVE if Bypass selected OR in Maintenance Mode,
   // or in Override Mode if Override Bypassing is configured.
   30: [XIC(Wrk_Bypass) OTE(Sts_Bypass) ,XIC(Sts_Maint) ,XIC(Sts_Ovrd) XIC(Cfg_OvrdPermIntlk) ]OTE(Sts_BypActive);
   // If a Maintenance Bypass function is active, display the Maintenance Bypass
   // Indicator (triangle symbol) on the graphic symbol.  Bypass functions are:
   // *  Interlock / Permissive Bypass function is enabled
   // *  Motor HAS run feedback designated by engineer, but
   // maintenance has selected to NOT USE run feedback
   31: [XIC(Sts_Bypass) ,XIC(Cfg_HasRunFdbk) XIO(Cfg_UseRunFdbk) ]OTE(Sts_MaintByp);
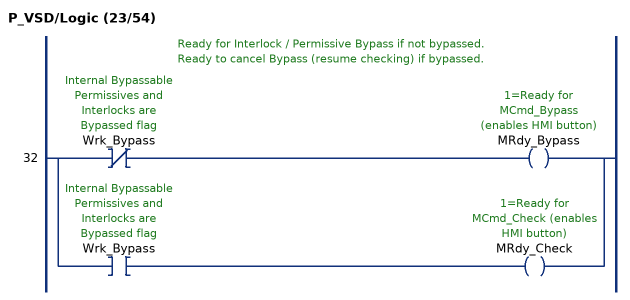
   // Ready for Interlock / Permissive Bypass if not bypassed.
   // Ready to cancel Bypass (resume checking) if bypassed.
   32: [XIO(Wrk_Bypass) OTE(MRdy_Bypass) ,XIC(Wrk_Bypass) OTE(MRdy_Check) ];
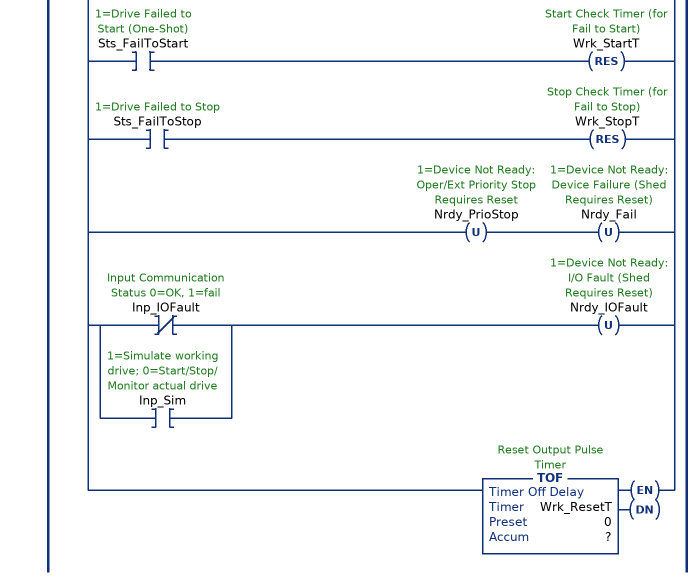
   // ============================================================
   // ALARM RESET COMMAND HANDLING
   // ============================================================
   // This rung handles the Alarm Reset Input and Commands
   // and the "Reset and Ack All" Operator Command.
   // This rung processes received Reset Commands from:
   // 1.  The Operator via HMI Operator Command, or
   // 2.  Higher-level strategies via Program Command
   // 3.  Pushbuttons or other block via Input
   // 4.  Resets initiated by other device Operator Commands (if configured to do so)
   // and forwards the Reset to ALL Alarms and latched Shed conditions.
   // The reset starts the Reset Timer (One-Shot Off-Delay)
   // to ensure the output is held on for at least the minimum time.
   // #####  V4.00.00  2018-07-13:  Deleted Cfg_PCmdClear; all Program Commands are now self-clearing.  #####
   // #####  Changed P_Mode to P_CmdSrc. Added External Command Source and Commands.  #####
   33: [XIC(OCmd_Reset) OTU(OCmd_Reset) ,XIC(XCmd_Reset) OTU(XCmd_Reset) ,XIC(PCmd_Reset) OTU(PCmd_Reset) ,XIC(Inp_Reset) ONS(Wrk_ResetONS) ,[XIC(OCmd_StartFwd) ,XIC(OCmd_StartRev) ,XIC(OCmd_Stop) ,[XIC(OCmd_JogFwd) ,XIC(OCmd_JogRev) ] XIC(Cfg_HasJog) ] XIC(Cfg_OCmdResets) XIC(Wrk_OperHas1) ,[XIC(XCmd_StartFwd) ,XIC(XCmd_StartRev) ,XIC(XCmd_Stop) ,[XIC(XCmd_JogFwd) ,XIC(XCmd_JogRev) ] XIC(Cfg_HasJog) ] XIC(Cfg_XCmdResets) XIC(Wrk_ExtHas1) ,XIC(OCmd_ResetAckAll) OTU(OCmd_ResetAckAll) [OTL(PCmd_FailToStartAck) ,OTL(PCmd_FailToStopAck) ,OTL(PCmd_DriveFaultAck) ,OTL(PCmd_IntlkTripAck) ,OTL(PCmd_IOFaultAck) ] ][OTL(FailToStart.PCmd_Reset) OTL(FailToStop.PCmd_Reset) OTL(IntlkTrip.PCmd_Reset) OTL(IOFault.PCmd_Reset) ,XIC(Sts_FailToStart) RES(Wrk_StartT) ,XIC(Sts_FailToStop) RES(Wrk_StopT) ,OTU(Nrdy_PrioStop) OTU(Nrdy_Fail) ,[XIO(Inp_IOFault) ,XIC(Inp_Sim) ] OTU(Nrdy_IOFault) ,TOF(Wrk_ResetT,?,?) ];
